(* CoDeSys 2.3.9.42 project: GLX_VCU_v3.3.0.pro *)
(* Author: JvL *)
(* Libraries: ifm_RAWCan\ifm_RAWCan_NT_V020004.lib 7.6.24 16:48:07, ifm_CR0403\ifm_CR0403_V030400.lib 31.5.24 17:04:27, ifm_CANopen\ifm_NetVarLib_NT_V020004.lib 7.6.24 16:46:42, standard.lib 4.10.05 11:14:46, SysLibCallback.lib 7.6.24 16:43:25, 3S_CANOPENNETVAR.LIB 7.6.24 16:46:41, Iecsfc.lib 13.4.06 15:51:28, Util.lib 7.6.24 16:43:26, ifm_CANopen\3S_CANopenManager.lib 7.6.24 16:46:41, ifm_CANopen\3S_CanDrv.lib 7.6.24 16:46:41 *)

(* PLC configuration (modules and I/O channels)
Configuration [LocalConfiguration] node 0, in %IB0 out %QB0 {IFM_PARAM_WORD_TIME = 0}
AT %IB0 [ChInputBool] Input 00 Bit
AT %IB1 [ChInputBool] Input 01 Bit
AT %IB2 [ChInputBool] Input 02 Bit
AT %IB3 [ChInputBool] Input 03 Bit
IGNITION_KEY AT %IB4 [ChInputBool] Input 04 Bit
CHARGER_INPUT AT %IB5 [ChInputBool] Input 05 Bit
BATTERY1_IGNITION AT %IB6 [ChInputBool] Input 06 Bit
BATTERY2_IGNITION AT %IB7 [ChInputBool] Input 07 Bit
ARM_SWITCH AT %IB8 [ChInputBool] Input 08 Bit
KILL_SWITCH AT %IB9 [ChInputBool] Input 09 Bit
HYDRAULIC_SWITCH AT %IB10 [ChInputBool] Input 10 Bit
EM_SWITCH AT %IB11 [ChInputBool] Input 11 Bit
ARM_LED AT %QB0 [ChOutputBool] Output 00 Bit
PRECHARGE_RELAY AT %QB1 [ChOutputBool] Output 01 Bit
AT %QB2 [ChOutputBool] Output 02 Bit
BRAKE_LIGHT AT %QB3 [ChOutputBool] Output 03 Bit
EM_BRAKE AT %QB4 [ChOutputBool] Output 04 Bit
MCU_IGNITION AT %QB5 [ChOutputBool] Output 05 Bit
BATTERY1_RELAY AT %QB6 [ChOutputBool] Output 06 Bit
BATTERY2_RELAY AT %QB7 [ChOutputBool] Output 07 Bit
HORN AT %QB8 [ChOutputBool] Output 08 Bit
BUZZER AT %QB9 [ChOutputBool] Output 09 Bit
CONTACTOR AT %QB10 [ChOutputBool] Output 10 Bit
CHARGING_LED AT %QB11 [ChOutputBool] Output 11 Bit
System Inputs [LocalSystemInputs] node 2, in %IB12 out %QB12
  SUPPLY_VOLTAGE_VBBS AT %IW6 [ChInputWord] Supply voltage VBBS
  SUPPLY_VOLTAGE_VU AT %IW7 [ChInputWord] Supply voltage VU
  SUPPLY_VOLTAGE_VBB1 AT %IW8 [ChInputWord] Supply voltage VBB1
  SUPPLY_VOLTAGE_VBB2 AT %IW9 [ChInputWord] Supply voltage VBB2
  TEMPERATURE AT %IW10 [ChInputInt] Temperature
J1939 Interface [CAN_J1939] node 1, in %IB37 out %QB12
Interface CAN 2 [CAN_BUS] node 1, in %IB37 out %QB12 {STACK_DWORD_S = 0}
  J1939 Interface [CAN_J1939] node 1, in %IB37 out %QB12
*)

(* Global variable list: CanOpen implicit Variables *)
VAR_GLOBAL CONSTANT
	MAX_CTRLINDEX : INT := 0;
END_VAR

(* Global variable list: Global_Variables *)
VAR_GLOBAL
(*BATTERY*)
	BATTERY1_SOC: BYTE;
	BATTERY1_SOH: BYTE;
	BATTERY1_CHARGING: BOOL;
	BATTERY1_POWER: INT;
	BATTERY1_NTC1: BYTE;
	BATTERY1_NTC2: BYTE;
	BATTERY1_CAN_ERROR: BOOL;
	BATTERY1_CAPACITY: INT;
	BATTERY1_TOTAL_CAPACITY: INT;
	BATTERY1_CURRENT: INT;
	BATTERY1_FULLCHARGE_MIN: REAL;

	BATTERY2_SOC: BYTE;
	BATTERY2_SOH: BYTE;
	BATTERY2_CHARGING: BOOL;
	BATTERY2_POWER: INT;
	BATTERY2_NTC1: BYTE;
	BATTERY2_NTC2: BYTE;
	BATTERY2_CAN_ERROR: BOOL;
	BATTERY2_CAPACITY: INT;
	BATTERY2_TOTAL_CAPACITY: INT;
	BATTERY2_CURRENT: INT;
	BATTERY2_FULLCHARGE_MIN: REAL;

(*MCU <> MOTOR*)
	MOTOR_TARGET_RPM: ARRAY [1..6] OF INT;
	MOTOR_IGNITION: ARRAY [1..6] OF BOOL;

	MOTOR_RPM: ARRAY [1..6] OF INT;
	MOTOR_POWER: ARRAY [1..6] OF INT;
	MOTOR_PHASE_CURRENT: ARRAY [1..6] OF WORD;
	MOTOR_TEMPERATURE:ARRAY [1..6] OF BYTE;
	MCU_TEMPERATURE:ARRAY [1..6] OF BYTE;
	MCU_CAN_ERROR: ARRAY [1..6] OF BOOL;

	MOTOR1_FAULT_ARRAY: ARRAY [1..4] OF BYTE;
	MOTOR2_FAULT_ARRAY: ARRAY [1..4] OF BYTE;
	MOTOR6_FAULT_ARRAY: ARRAY [1..4] OF BYTE;
       MOTOR_OBD_ARRAY: ARRAY [1..6] OF WORD;

(*JOYSTICK*)
	LOG_JX: BYTE;
	LOG_JY: BYTE;
	JOY_ERROR: BOOL;
(*IMU*)
	X_ANGLE_BYTE:BYTE;
	Y_ANGLE_BYTE:BYTE;
	NEG_Y: BOOL;
	NEG_X: BOOL;
	Y_MAX_PEAK: BYTE;
	X_MAX_PEAK: BYTE;
	Y_MIN_PEAK: BYTE;
	X_MIN_PEAK: BYTE;
	IMU_CAN_ERROR:BOOL;
	IMU_ALERT: BOOL;
(*DISPLAY TELEMATICS*)
	HIGH_SPEED: BOOL;
	POWER_MODE: BOOL;
	HILL_HOLD: BOOL;
	DISABLE_MCU_CAN: BOOL;
	TRIP_RESET: BOOL;
      	BATTERY_CHARGING:BOOL;
(*MISC*)
	REVERSE: BOOL;
	MCU_BRAKE: BOOL;
(*HYDRAULICS*)
	HYDRAULIC_IGNITION: BOOL;
(*CALCULATIONS*)
	AVG_RPM: INT;
	RANGE_IN_KM: BYTE;
	SPEED: BYTE;

	RUNTIME: DWORD;
	HYDL_UP_TIME:DWORD;
	VEHICLE_UP_TIME: DWORD;
	VEHICLE_UP_TIME_LT: DWORD;

	ODO_KM: WORD;
	ODO_METER: DWORD;

	TRIP_METER: DWORD;
	TRIP_KM: WORD;

	DUMMY: BOOL;
END_VAR
VAR_GLOBAL RETAIN
	Y_MAX_RETAIN: BYTE;
	X_MAX_RETAIN: BYTE;
	Y_MIN_RETAIN: BYTE;
	X_MIN_RETAIN: BYTE;
END_VAR

(* Global variable list: Networkmanagement implicit Variables CAN *)
VAR_GLOBAL CONSTANT
	USE_NWVARS_CAN : BOOL := FALSE;
	MAX_NetVarItems_CAN	: INT := 0;
	MAX_NetVarPDO_Rx_CAN	: INT := 0;
	MAX_NetVarPDO_Tx_CAN	: INT := 0;
	MAX_NetVarOD_CAN		: INT := 0;
END_VAR
VAR_GLOBAL
	pNetVarItems_CAN		: ARRAY[0..MAX_NetVarItems_CAN] OF NetVarDataItem_CAN;
	pNetVarPDO_Rx_CAN		: ARRAY[0..MAX_NetVarPDO_Rx_CAN] OF NetVarPDO_Rx_CAN;
	pNetVarPDO_Tx_CAN		: ARRAY[0..MAX_NetVarPDO_Tx_CAN] OF NetVarPDO_Tx_CAN;
	pNetVarOD_CAN			: ARRAY[0..MAX_NetVarOD_CAN] OF NetVarOD_CAN;
END_VAR

(* POU PLC_PRG, FBD *)
PROGRAM PLC_PRG
VAR
	CONTACTOR_DELAY: TON;
END_VAR
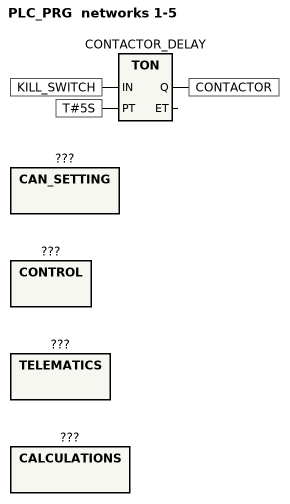
_FBD_ (* Function Block Diagram *)
NETWORK 1
	CONTACTOR_DELAY:TON(IN: KILL_SWITCH, PT: T#5S) => CONTACTOR
NETWORK 2
	???:CAN_SETTING()
NETWORK 3
	???:CONTROL()
NETWORK 4
	???:TELEMATICS()
NETWORK 5
	???:CALCULATIONS()
_END_FBD_
(* the same logic as Structured Text *)
(* Network 1 *)
CONTACTOR_DELAY(IN := KILL_SWITCH, PT := T#5S);
CONTACTOR := CONTACTOR_DELAY.Q;
(* Network 2: see the listing above *)
(* Network 3: see the listing above *)
(* Network 4: see the listing above *)
(* Network 5: see the listing above *)
END_PROGRAM

(* POU CAN_SETTING/CAN_SETTING, FBD *)
PROGRAM CAN_SETTING
(*
Created By: BHAGYESH
Date: 20-01-2024
Version: 1
Description: This program enables the CAN channels and sets the basic CAN parameter for both channels.
This block also controls the IFM's Inbuilt LED.
*)
VAR
	CAN_EN_1: CAN_ENABLE;
	CAN_EN_2: CAN_ENABLE;
	CAN_SET_1: CAN_SETDOWNLOADID;
	CAN_SET_2: CAN_SETDOWNLOADID;
	LED_SET: SET_LED;
	CAN_STATUS_1: CAN_STATUS;
	CAN_STATUS_2: CAN_STATUS;
	RESET_1: BOOL;
	RESET_2: BOOL;
END_VAR
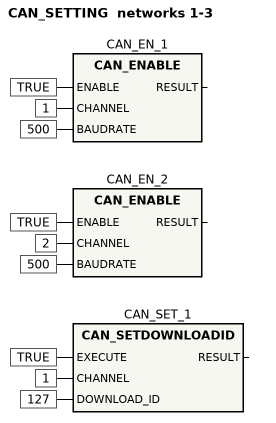
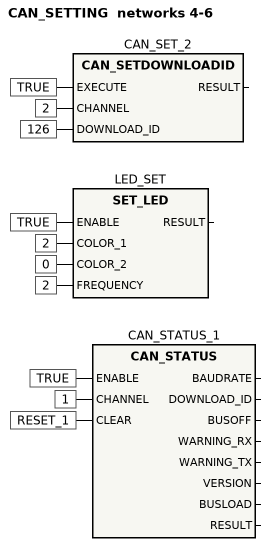
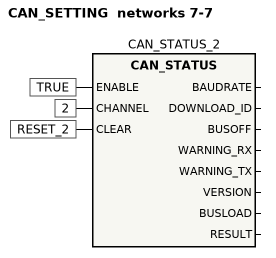
_FBD_ (* Function Block Diagram *)
NETWORK 1
	CAN_EN_1:CAN_ENABLE(ENABLE: TRUE, CHANNEL: 1, BAUDRATE: 500)
NETWORK 2
	CAN_EN_2:CAN_ENABLE(ENABLE: TRUE, CHANNEL: 2, BAUDRATE: 500)
NETWORK 3
	CAN_SET_1:CAN_SETDOWNLOADID(EXECUTE: TRUE, CHANNEL: 1, DOWNLOAD_ID: 127)
NETWORK 4
	CAN_SET_2:CAN_SETDOWNLOADID(EXECUTE: TRUE, CHANNEL: 2, DOWNLOAD_ID: 126)
NETWORK 5
	LED_SET:SET_LED(ENABLE: TRUE, COLOR_1: 2, COLOR_2: 0, FREQUENCY: 2)
NETWORK 6
	CAN_STATUS_1:CAN_STATUS(ENABLE: TRUE, CHANNEL: 1, CLEAR: RESET_1)
NETWORK 7
	CAN_STATUS_2:CAN_STATUS(ENABLE: TRUE, CHANNEL: 2, CLEAR: RESET_2)
_END_FBD_
(* the same logic as Structured Text *)
(* Network 1 *)
CAN_EN_1(ENABLE := TRUE, CHANNEL := 1, BAUDRATE := 500);
(* Network 2 *)
CAN_EN_2(ENABLE := TRUE, CHANNEL := 2, BAUDRATE := 500);
(* Network 3 *)
CAN_SET_1(EXECUTE := TRUE, CHANNEL := 1, DOWNLOAD_ID := 127);
(* Network 4 *)
CAN_SET_2(EXECUTE := TRUE, CHANNEL := 2, DOWNLOAD_ID := 126);
(* Network 5 *)
LED_SET(ENABLE := TRUE, COLOR_1 := 2, COLOR_2 := 0, FREQUENCY := 2);
(* Network 6 *)
CAN_STATUS_1(ENABLE := TRUE, CHANNEL := 1, CLEAR := RESET_1);
(* Network 7 *)
CAN_STATUS_2(ENABLE := TRUE, CHANNEL := 2, CLEAR := RESET_2);
END_PROGRAM

(* POU CONTROL, LD *)
PROGRAM CONTROL
(*
CH1 (500KBPS) :  MAKERSAN JOYSTICK								CH2 (500KBPS):	CLN BATTERY1
					DWIN DISPLAY															CLN BATTERY2
					BYTEBEAM  &  TOR														CHARA MCU 1
					MAKESAN IMU															CHARA MCU 2	
																								CHARA MCU 3
																								SOLTERRA CHARGER
			***UPDATES***
> Visualization update
> Chara can tx block updated
> Actual rpm of tx block changed to reference rpm
>Updated AVG_RPM in tx block input.
> MAKERSAN Joystick added
>RPM FACTOR IS 40 for 4000 RPM
> Battery channel changed and ramp decreased
>BATTERY CHARGING 
>MCU HIGH TEMP CUTOFF
>SALERI PUMP 
>HIGH SPEED AND HORN BUTTON INVRTED

>The MCU has min ramp time of 100ms.
*)
VAR
	BATTERY: CLN_BATTERY;
	BATTERY_SELECTION: CLN_BATTERY_SELECTION;
	AUTO_CHARGING: CLN_CHARGING;

	JOYSTICK: MAKERSAN_JOYSTICK;
	ALT_SPEED: ALTERNATE;
	IMU: IMU_SENSOR;
	HYDRAULICS: HYDRAULIC_CONTROL;
	ARM: ARM_LOGIC;

	DRIVE: DRIVE_LOGIC;
	THROTTLE: THROTTLE_LOGIC;
	THROTTLE_RIGHT: INT;
	THROTTLE_LEFT: INT;

	MCU_TX_RIGHT: CHARA_MCU_TX;
	MCU_TX_LEFT: CHARA_MCU_TX;
	MCU_RX_RIGHT: CHARA_MCU_RX;
	MCU_RX_LEFT: CHARA_MCU_RX;

	SALERI_PUMP: PWM1000;
	COOLANT_PUMP_ON: BOOL;
      VAL:WORD;

	RIGHT_ZERO: BOOL;
	LEFT_ZERO: BOOL;
	POWER_ZERO: BOOL;

	TEMP_CUTOFF: BOOL;
	MCU_HIGH_TEMP: BOOL;
	MCU_LOW_TEMP: BOOL;

	LOW5_SOC: BOOL;
	LOW20_SOC: BOOL;
	LOW_SOC: F_TRIG;
	LOW_SOC_TIMER: TP;
	LOWSOC_BLINK: BLINK;

	IMU_BLINK: BLINK;
	REVERSE_BLINK: BLINK;
	CHARGE_ERROR_BLINK: BLINK;
       LOW_SOC_BUZZER: BOOL;

	RX_227: RX_CAN;
	TOF_227: TOF;
	CHARGER_5kW_INPUT: BOOL;
	CHARGING_5KW: CAN_TX;

	CHARGE_ERROR_LIGHT: BLINK;
	DDD: BOOL;
	STARTING_BLINK: BLINK;
	OVER_TEMP_BLINK: BLINK;
END_VAR
VAR CONSTANT
	RPM_FACTOR: INT := 45;
	RAMP: INT:= 1000;
	MCU_RAMP: BYTE := 8;
	PHASE_LIMIT: BYTE := 60;
	CHARGING_FRAME: ARRAY [0..7] OF BYTE := 16#03, 16#25, 16#01, 16#90, 0, 0, 0, 0;
END_VAR
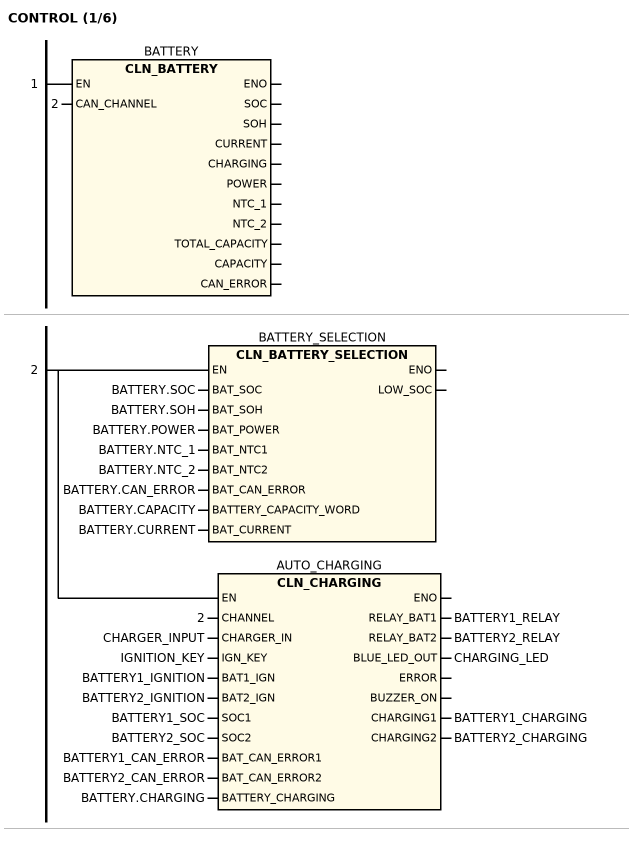
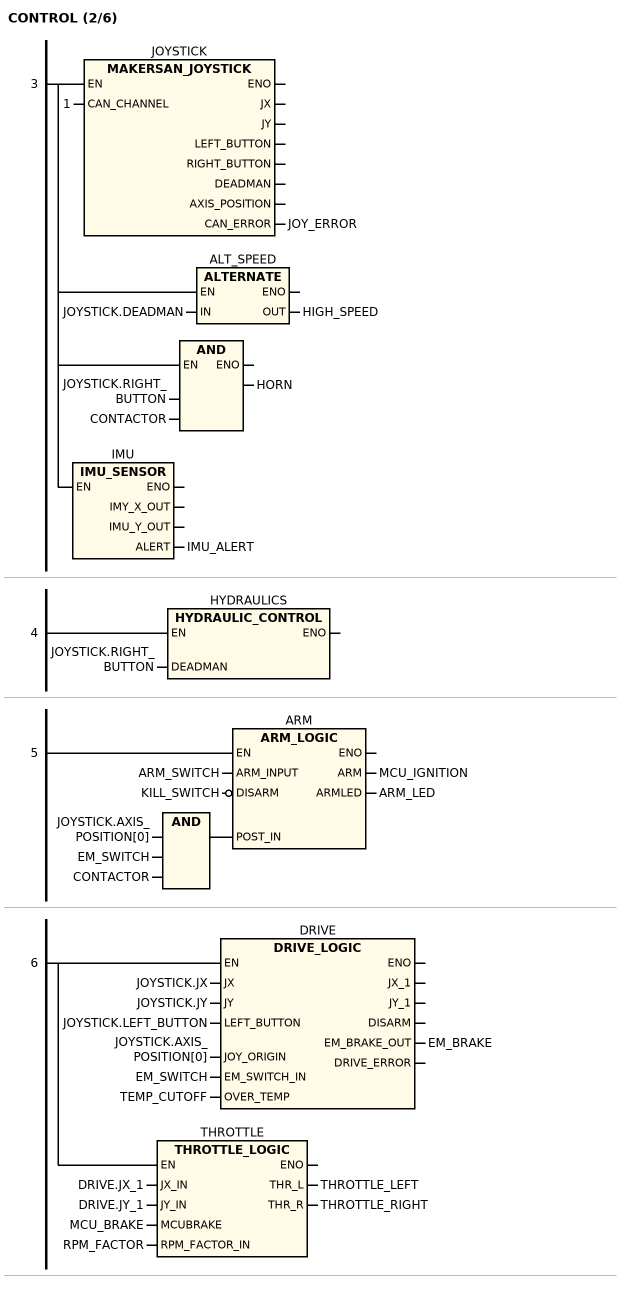
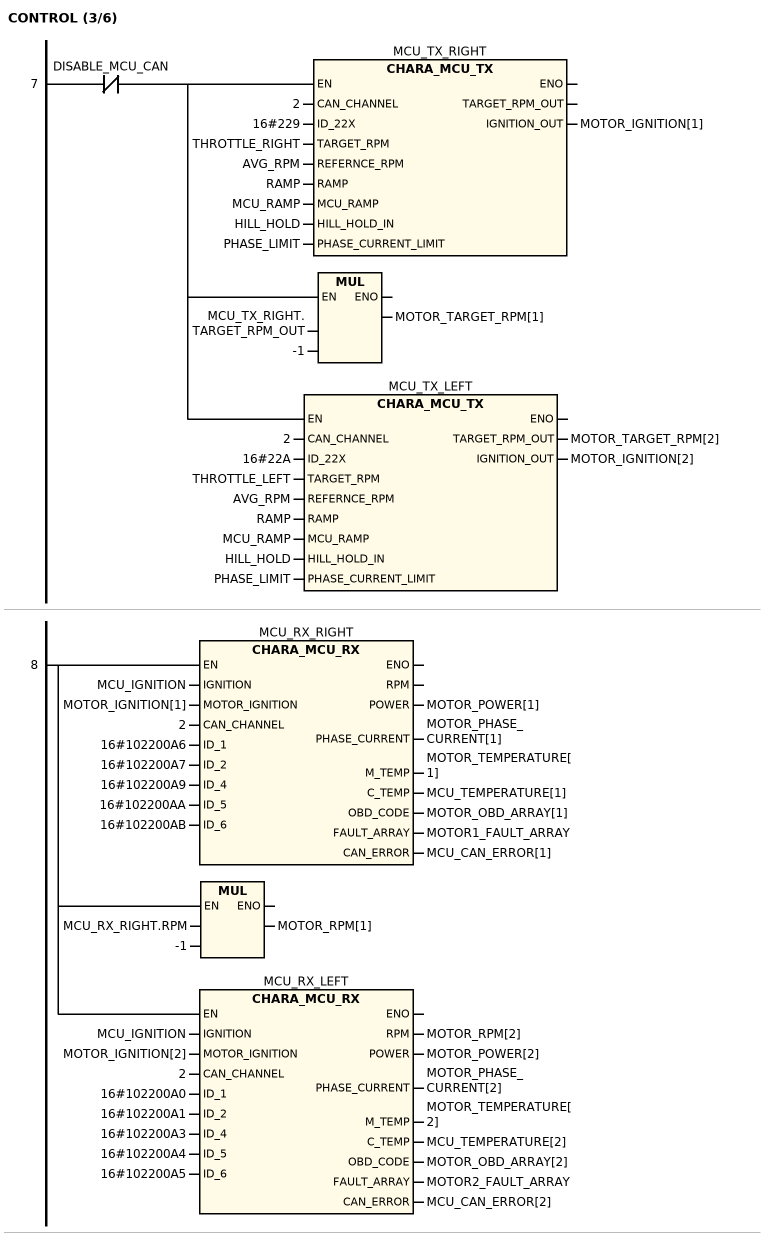
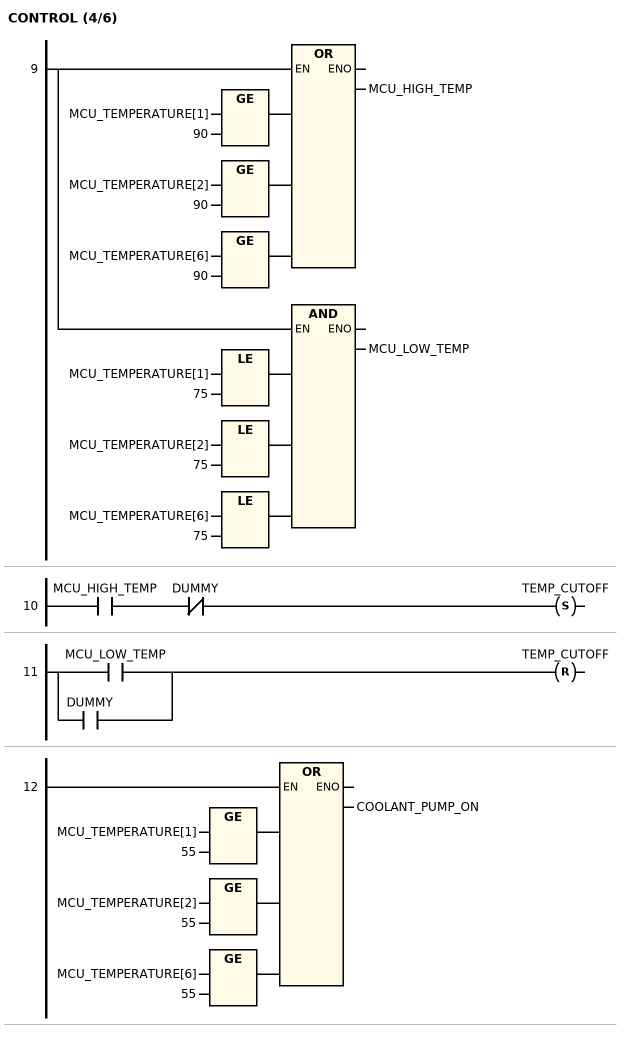
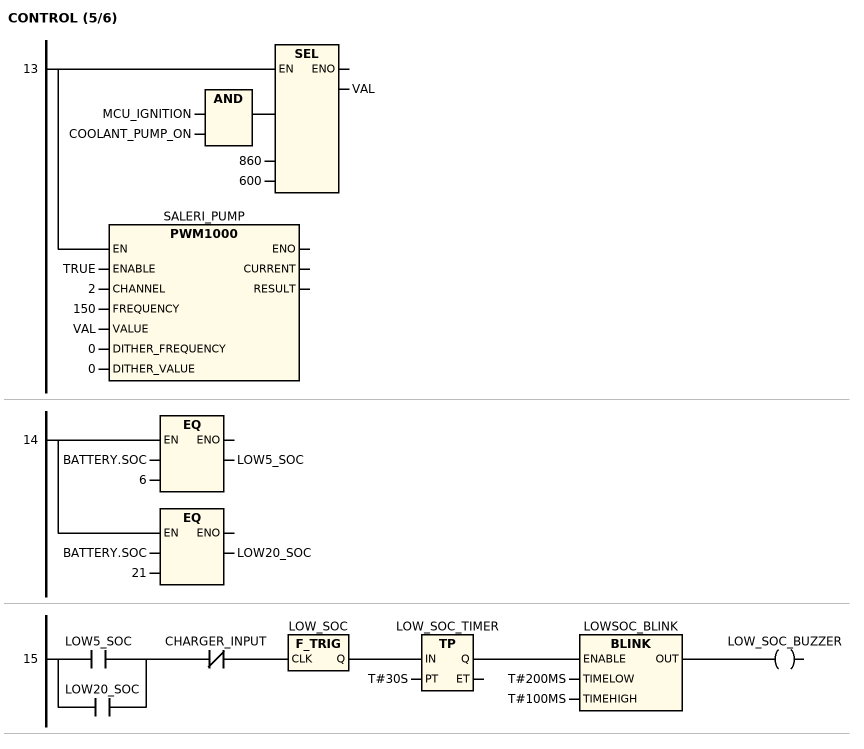
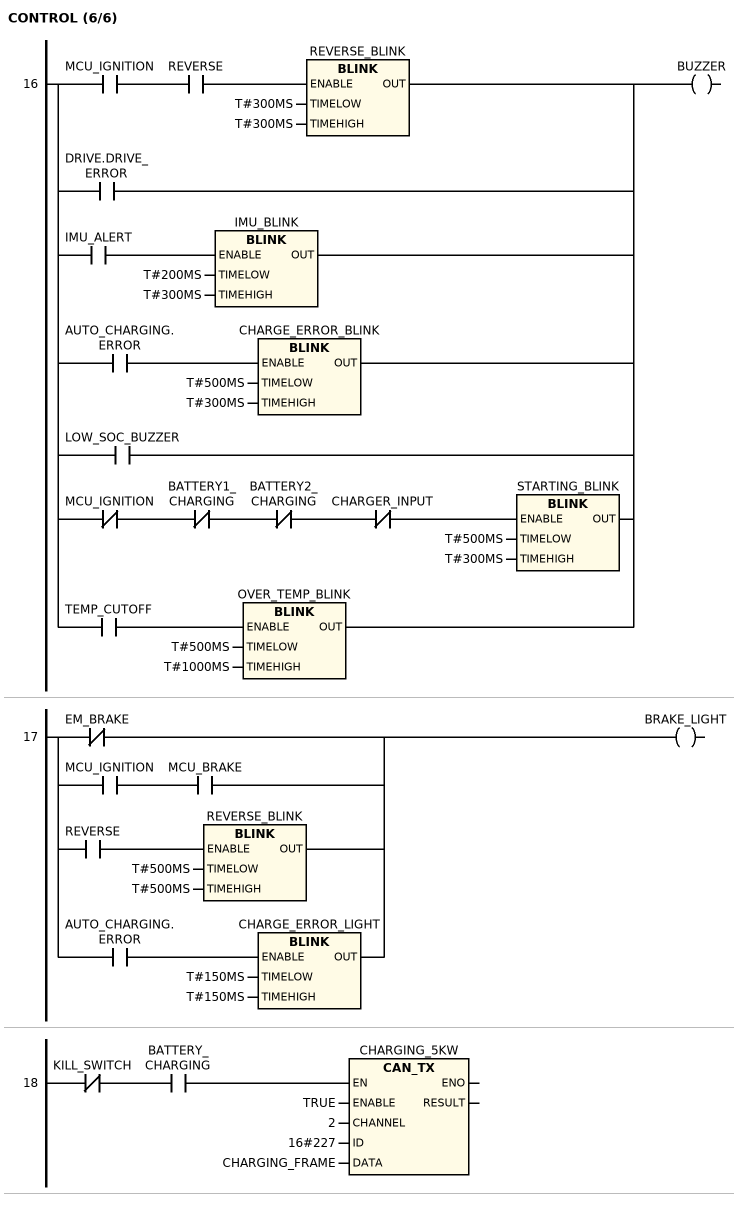
_LD_ (* Ladder Diagram *)
NETWORK 1
	*
		EN --- BATTERY:CLN_BATTERY(CAN_CHANNEL: 2)
NETWORK 2
	*
		EN --- BATTERY_SELECTION:CLN_BATTERY_SELECTION(BAT_SOC: BATTERY.SOC, BAT_SOH: BATTERY.SOH, BAT_POWER: BATTERY.POWER, BAT_NTC1: BATTERY.NTC_1, BAT_NTC2: BATTERY.NTC_2, BAT_CAN_ERROR: BATTERY.CAN_ERROR, BATTERY_CAPACITY_WORD: BATTERY.CAPACITY, BAT_CURRENT: BATTERY.CURRENT)
		EN --- AUTO_CHARGING:CLN_CHARGING(CHANNEL: 2, CHARGER_IN: CHARGER_INPUT, IGN_KEY: IGNITION_KEY, BAT1_IGN: BATTERY1_IGNITION, BAT2_IGN: BATTERY2_IGNITION, SOC1: BATTERY1_SOC, SOC2: BATTERY2_SOC, BAT_CAN_ERROR1: BATTERY1_CAN_ERROR, BAT_CAN_ERROR2: BATTERY2_CAN_ERROR, BATTERY_CHARGING: BATTERY.CHARGING, RELAY_BAT2 => BATTERY2_RELAY, BLUE_LED_OUT => CHARGING_LED, CHARGING1 => BATTERY1_CHARGING, CHARGING2 => BATTERY2_CHARGING) => BATTERY1_RELAY
NETWORK 3
	*
		EN --- JOYSTICK:MAKERSAN_JOYSTICK(CAN_CHANNEL: 1, CAN_ERROR => JOY_ERROR)
		EN --- ALT_SPEED:ALTERNATE(IN: JOYSTICK.DEADMAN) => HIGH_SPEED
		EN --- AND(JOYSTICK.RIGHT_BUTTON, CONTACTOR) => HORN
		EN --- IMU:IMU_SENSOR(ALERT => IMU_ALERT)
NETWORK 4
	*
		EN --- HYDRAULICS:HYDRAULIC_CONTROL(DEADMAN: JOYSTICK.RIGHT_BUTTON)
NETWORK 5
	*
		EN --- ARM:ARM_LOGIC(ARM_INPUT: ARM_SWITCH, DISARM: NOT KILL_SWITCH, POST_IN: AND(JOYSTICK.AXIS_POSITION[0], EM_SWITCH, CONTACTOR), ARMLED => ARM_LED) => MCU_IGNITION
NETWORK 6
	*
		EN --- DRIVE:DRIVE_LOGIC(JX: JOYSTICK.JX, JY: JOYSTICK.JY, LEFT_BUTTON: JOYSTICK.LEFT_BUTTON, JOY_ORIGIN: JOYSTICK.AXIS_POSITION[0], EM_SWITCH_IN: EM_SWITCH, OVER_TEMP: TEMP_CUTOFF, EM_BRAKE_OUT => EM_BRAKE)
		EN --- THROTTLE:THROTTLE_LOGIC(JX_IN: DRIVE.JX_1, JY_IN: DRIVE.JY_1, MCUBRAKE: MCU_BRAKE, RPM_FACTOR_IN: RPM_FACTOR, THR_R => THROTTLE_RIGHT) => THROTTLE_LEFT
NETWORK 7
	[/DISABLE_MCU_CAN]
		EN --- MCU_TX_RIGHT:CHARA_MCU_TX(CAN_CHANNEL: 2, ID_22X: 16#229, TARGET_RPM: THROTTLE_RIGHT, REFERNCE_RPM: AVG_RPM, RAMP: RAMP, MCU_RAMP: MCU_RAMP, HILL_HOLD_IN: HILL_HOLD, PHASE_CURRENT_LIMIT: PHASE_LIMIT, IGNITION_OUT => MOTOR_IGNITION[1])
		EN --- MUL(MCU_TX_RIGHT.TARGET_RPM_OUT, -1) => MOTOR_TARGET_RPM[1]
		EN --- MCU_TX_LEFT:CHARA_MCU_TX(CAN_CHANNEL: 2, ID_22X: 16#22A, TARGET_RPM: THROTTLE_LEFT, REFERNCE_RPM: AVG_RPM, RAMP: RAMP, MCU_RAMP: MCU_RAMP, HILL_HOLD_IN: HILL_HOLD, PHASE_CURRENT_LIMIT: PHASE_LIMIT, IGNITION_OUT => MOTOR_IGNITION[2]) => MOTOR_TARGET_RPM[2]
NETWORK 8
	*
		EN --- MCU_RX_RIGHT:CHARA_MCU_RX(IGNITION: MCU_IGNITION, MOTOR_IGNITION: MOTOR_IGNITION[1], CAN_CHANNEL: 2, ID_1: 16#102200A6, ID_2: 16#102200A7, ID_4: 16#102200A9, ID_5: 16#102200AA, ID_6: 16#102200AB, POWER => MOTOR_POWER[1], PHASE_CURRENT => MOTOR_PHASE_CURRENT[1], M_TEMP => MOTOR_TEMPERATURE[1], C_TEMP => MCU_TEMPERATURE[1], OBD_CODE => MOTOR_OBD_ARRAY[1], FAULT_ARRAY => MOTOR1_FAULT_ARRAY, CAN_ERROR => MCU_CAN_ERROR[1])
		EN --- MUL(MCU_RX_RIGHT.RPM, -1) => MOTOR_RPM[1]
		EN --- MCU_RX_LEFT:CHARA_MCU_RX(IGNITION: MCU_IGNITION, MOTOR_IGNITION: MOTOR_IGNITION[2], CAN_CHANNEL: 2, ID_1: 16#102200A0, ID_2: 16#102200A1, ID_4: 16#102200A3, ID_5: 16#102200A4, ID_6: 16#102200A5, POWER => MOTOR_POWER[2], PHASE_CURRENT => MOTOR_PHASE_CURRENT[2], M_TEMP => MOTOR_TEMPERATURE[2], C_TEMP => MCU_TEMPERATURE[2], OBD_CODE => MOTOR_OBD_ARRAY[2], FAULT_ARRAY => MOTOR2_FAULT_ARRAY, CAN_ERROR => MCU_CAN_ERROR[2]) => MOTOR_RPM[2]
NETWORK 9
	*
		EN --- OR(GE(MCU_TEMPERATURE[1], 90), GE(MCU_TEMPERATURE[2], 90), GE(MCU_TEMPERATURE[6], 90)) => MCU_HIGH_TEMP
		EN --- AND(LE(MCU_TEMPERATURE[1], 75), LE(MCU_TEMPERATURE[2], 75), LE(MCU_TEMPERATURE[6], 75)) => MCU_LOW_TEMP
NETWORK 10
	[MCU_HIGH_TEMP] - [/DUMMY] --- (S TEMP_CUTOFF)
NETWORK 11
	{ [MCU_LOW_TEMP] | [DUMMY] } --- (R TEMP_CUTOFF)
NETWORK 12
	*
		EN --- OR(GE(MCU_TEMPERATURE[1], 55), GE(MCU_TEMPERATURE[2], 55), GE(MCU_TEMPERATURE[6], 55)) => COOLANT_PUMP_ON
NETWORK 13
	*
		EN --- SEL(AND(MCU_IGNITION, COOLANT_PUMP_ON), 860, 600) => VAL
		EN --- SALERI_PUMP:PWM1000(ENABLE: TRUE, CHANNEL: 2, FREQUENCY: 150, VALUE: VAL, DITHER_FREQUENCY: 0, DITHER_VALUE: 0)
NETWORK 14
	*
		EN --- EQ(BATTERY.SOC, 6) => LOW5_SOC
		EN --- EQ(BATTERY.SOC, 21) => LOW20_SOC
NETWORK 15
	{ [LOW5_SOC] | [LOW20_SOC] } - [/CHARGER_INPUT] - LOW_SOC:F_TRIG(CLK: *) - LOW_SOC_TIMER:TP(IN: *, PT: T#30S) - LOWSOC_BLINK:BLINK(ENABLE: *, TIMELOW: T#200MS, TIMEHIGH: T#100MS) --- (LOW_SOC_BUZZER)
NETWORK 16
	{ [MCU_IGNITION] - [REVERSE] - REVERSE_BLINK:BLINK(ENABLE: *, TIMELOW: T#300MS, TIMEHIGH: T#300MS) | [DRIVE.DRIVE_ERROR] | [IMU_ALERT] - IMU_BLINK:BLINK(ENABLE: *, TIMELOW: T#200MS, TIMEHIGH: T#300MS) | [AUTO_CHARGING.ERROR] - CHARGE_ERROR_BLINK:BLINK(ENABLE: *, TIMELOW: T#500MS, TIMEHIGH: T#300MS) | [LOW_SOC_BUZZER] | [/MCU_IGNITION] - [/BATTERY1_CHARGING] - [/BATTERY2_CHARGING] - [/CHARGER_INPUT] - STARTING_BLINK:BLINK(ENABLE: *, TIMELOW: T#500MS, TIMEHIGH: T#300MS) | [TEMP_CUTOFF] - OVER_TEMP_BLINK:BLINK(ENABLE: *, TIMELOW: T#500MS, TIMEHIGH: T#1000MS) } --- (BUZZER)
NETWORK 17
	{ [/EM_BRAKE] | [MCU_IGNITION] - [MCU_BRAKE] | [REVERSE] - REVERSE_BLINK:BLINK(ENABLE: *, TIMELOW: T#500MS, TIMEHIGH: T#500MS) | [AUTO_CHARGING.ERROR] - CHARGE_ERROR_LIGHT:BLINK(ENABLE: *, TIMELOW: T#150MS, TIMEHIGH: T#150MS) } --- (BRAKE_LIGHT)
NETWORK 18
	[/KILL_SWITCH] - [BATTERY_CHARGING]
		EN --- CHARGING_5KW:CAN_TX(ENABLE: TRUE, CHANNEL: 2, ID: 16#227, DATA: CHARGING_FRAME)
_END_LD_
(* the same logic as Structured Text *)
(* Network 1 *)
BATTERY(CAN_CHANNEL := 2);
(* Network 2 *)
BATTERY_SELECTION(BAT_SOC := BATTERY.SOC, BAT_SOH := BATTERY.SOH, BAT_POWER := BATTERY.POWER, BAT_NTC1 := BATTERY.NTC_1, BAT_NTC2 := BATTERY.NTC_2, BAT_CAN_ERROR := BATTERY.CAN_ERROR, BATTERY_CAPACITY_WORD := BATTERY.CAPACITY, BAT_CURRENT := BATTERY.CURRENT);
AUTO_CHARGING(CHANNEL := 2, CHARGER_IN := CHARGER_INPUT, IGN_KEY := IGNITION_KEY, BAT1_IGN := BATTERY1_IGNITION, BAT2_IGN := BATTERY2_IGNITION, SOC1 := BATTERY1_SOC, SOC2 := BATTERY2_SOC, BAT_CAN_ERROR1 := BATTERY1_CAN_ERROR, BAT_CAN_ERROR2 := BATTERY2_CAN_ERROR, BATTERY_CHARGING := BATTERY.CHARGING);
BATTERY2_RELAY := AUTO_CHARGING.RELAY_BAT2;
CHARGING_LED := AUTO_CHARGING.BLUE_LED_OUT;
BATTERY1_CHARGING := AUTO_CHARGING.CHARGING1;
BATTERY2_CHARGING := AUTO_CHARGING.CHARGING2;
BATTERY1_RELAY := AUTO_CHARGING.RELAY_BAT1;
(* Network 3 *)
JOYSTICK(CAN_CHANNEL := 1);
JOY_ERROR := JOYSTICK.CAN_ERROR;
ALT_SPEED(IN := JOYSTICK.DEADMAN);
HIGH_SPEED := ALT_SPEED.OUT;
HORN := JOYSTICK.RIGHT_BUTTON AND CONTACTOR;
IMU();
IMU_ALERT := IMU.ALERT;
(* Network 4 *)
HYDRAULICS(DEADMAN := JOYSTICK.RIGHT_BUTTON);
(* Network 5 *)
ARM(ARM_INPUT := ARM_SWITCH, DISARM := NOT KILL_SWITCH, POST_IN := JOYSTICK.AXIS_POSITION[0] AND EM_SWITCH AND CONTACTOR);
ARM_LED := ARM.ARMLED;
MCU_IGNITION := ARM.ARM;
(* Network 6 *)
DRIVE(JX := JOYSTICK.JX, JY := JOYSTICK.JY, LEFT_BUTTON := JOYSTICK.LEFT_BUTTON, JOY_ORIGIN := JOYSTICK.AXIS_POSITION[0], EM_SWITCH_IN := EM_SWITCH, OVER_TEMP := TEMP_CUTOFF);
EM_BRAKE := DRIVE.EM_BRAKE_OUT;
THROTTLE(JX_IN := DRIVE.JX_1, JY_IN := DRIVE.JY_1, MCUBRAKE := MCU_BRAKE, RPM_FACTOR_IN := RPM_FACTOR);
THROTTLE_RIGHT := THROTTLE.THR_R;
THROTTLE_LEFT := THROTTLE.THR_L;
(* Network 7 *)
IF NOT DISABLE_MCU_CAN THEN
	MCU_TX_RIGHT(CAN_CHANNEL := 2, ID_22X := 16#229, TARGET_RPM := THROTTLE_RIGHT, REFERNCE_RPM := AVG_RPM, RAMP := RAMP, MCU_RAMP := MCU_RAMP, HILL_HOLD_IN := HILL_HOLD, PHASE_CURRENT_LIMIT := PHASE_LIMIT);
	MOTOR_IGNITION[1] := MCU_TX_RIGHT.IGNITION_OUT;
	MOTOR_TARGET_RPM[1] := MCU_TX_RIGHT.TARGET_RPM_OUT * (-1);
	MCU_TX_LEFT(CAN_CHANNEL := 2, ID_22X := 16#22A, TARGET_RPM := THROTTLE_LEFT, REFERNCE_RPM := AVG_RPM, RAMP := RAMP, MCU_RAMP := MCU_RAMP, HILL_HOLD_IN := HILL_HOLD, PHASE_CURRENT_LIMIT := PHASE_LIMIT);
	MOTOR_IGNITION[2] := MCU_TX_LEFT.IGNITION_OUT;
	MOTOR_TARGET_RPM[2] := MCU_TX_LEFT.TARGET_RPM_OUT;
END_IF;
(* Network 8 *)
MCU_RX_RIGHT(IGNITION := MCU_IGNITION, MOTOR_IGNITION := MOTOR_IGNITION[1], CAN_CHANNEL := 2, ID_1 := 16#102200A6, ID_2 := 16#102200A7, ID_4 := 16#102200A9, ID_5 := 16#102200AA, ID_6 := 16#102200AB);
MOTOR_POWER[1] := MCU_RX_RIGHT.POWER;
MOTOR_PHASE_CURRENT[1] := MCU_RX_RIGHT.PHASE_CURRENT;
MOTOR_TEMPERATURE[1] := MCU_RX_RIGHT.M_TEMP;
MCU_TEMPERATURE[1] := MCU_RX_RIGHT.C_TEMP;
MOTOR_OBD_ARRAY[1] := MCU_RX_RIGHT.OBD_CODE;
MOTOR1_FAULT_ARRAY := MCU_RX_RIGHT.FAULT_ARRAY;
MCU_CAN_ERROR[1] := MCU_RX_RIGHT.CAN_ERROR;
MOTOR_RPM[1] := MCU_RX_RIGHT.RPM * (-1);
MCU_RX_LEFT(IGNITION := MCU_IGNITION, MOTOR_IGNITION := MOTOR_IGNITION[2], CAN_CHANNEL := 2, ID_1 := 16#102200A0, ID_2 := 16#102200A1, ID_4 := 16#102200A3, ID_5 := 16#102200A4, ID_6 := 16#102200A5);
MOTOR_POWER[2] := MCU_RX_LEFT.POWER;
MOTOR_PHASE_CURRENT[2] := MCU_RX_LEFT.PHASE_CURRENT;
MOTOR_TEMPERATURE[2] := MCU_RX_LEFT.M_TEMP;
MCU_TEMPERATURE[2] := MCU_RX_LEFT.C_TEMP;
MOTOR_OBD_ARRAY[2] := MCU_RX_LEFT.OBD_CODE;
MOTOR2_FAULT_ARRAY := MCU_RX_LEFT.FAULT_ARRAY;
MCU_CAN_ERROR[2] := MCU_RX_LEFT.CAN_ERROR;
MOTOR_RPM[2] := MCU_RX_LEFT.RPM;
(* Network 9 *)
MCU_HIGH_TEMP := (MCU_TEMPERATURE[1] >= 90) OR (MCU_TEMPERATURE[2] >= 90) OR (MCU_TEMPERATURE[6] >= 90);
MCU_LOW_TEMP := (MCU_TEMPERATURE[1] <= 75) AND (MCU_TEMPERATURE[2] <= 75) AND (MCU_TEMPERATURE[6] <= 75);
(* Network 10 *)
IF MCU_HIGH_TEMP AND NOT DUMMY THEN TEMP_CUTOFF := TRUE; END_IF;
(* Network 11 *)
IF MCU_LOW_TEMP OR DUMMY THEN TEMP_CUTOFF := FALSE; END_IF;
(* Network 12 *)
COOLANT_PUMP_ON := (MCU_TEMPERATURE[1] >= 55) OR (MCU_TEMPERATURE[2] >= 55) OR (MCU_TEMPERATURE[6] >= 55);
(* Network 13 *)
VAL := SEL(MCU_IGNITION AND COOLANT_PUMP_ON, 860, 600);
SALERI_PUMP(ENABLE := TRUE, CHANNEL := 2, FREQUENCY := 150, VALUE := VAL, DITHER_FREQUENCY := 0, DITHER_VALUE := 0);
(* Network 14 *)
LOW5_SOC := BATTERY.SOC = 6;
LOW20_SOC := BATTERY.SOC = 21;
(* Network 15 *)
LOW_SOC(CLK := (LOW5_SOC OR LOW20_SOC) AND NOT CHARGER_INPUT);
LOW_SOC_TIMER(IN := LOW_SOC.Q, PT := T#30S);
LOWSOC_BLINK(ENABLE := LOW_SOC_TIMER.Q, TIMELOW := T#200MS, TIMEHIGH := T#100MS);
LOW_SOC_BUZZER := LOWSOC_BLINK.OUT;
(* Network 16 *)
REVERSE_BLINK(ENABLE := MCU_IGNITION AND REVERSE, TIMELOW := T#300MS, TIMEHIGH := T#300MS);
IMU_BLINK(ENABLE := IMU_ALERT, TIMELOW := T#200MS, TIMEHIGH := T#300MS);
CHARGE_ERROR_BLINK(ENABLE := AUTO_CHARGING.ERROR, TIMELOW := T#500MS, TIMEHIGH := T#300MS);
STARTING_BLINK(ENABLE := NOT MCU_IGNITION AND NOT BATTERY1_CHARGING AND NOT BATTERY2_CHARGING AND NOT CHARGER_INPUT, TIMELOW := T#500MS, TIMEHIGH := T#300MS);
OVER_TEMP_BLINK(ENABLE := TEMP_CUTOFF, TIMELOW := T#500MS, TIMEHIGH := T#1000MS);
BUZZER := REVERSE_BLINK.OUT OR DRIVE.DRIVE_ERROR OR IMU_BLINK.OUT OR CHARGE_ERROR_BLINK.OUT OR LOW_SOC_BUZZER OR STARTING_BLINK.OUT OR OVER_TEMP_BLINK.OUT;
(* Network 17 *)
REVERSE_BLINK(ENABLE := REVERSE, TIMELOW := T#500MS, TIMEHIGH := T#500MS);
CHARGE_ERROR_LIGHT(ENABLE := AUTO_CHARGING.ERROR, TIMELOW := T#150MS, TIMEHIGH := T#150MS);
BRAKE_LIGHT := NOT EM_BRAKE OR MCU_IGNITION AND MCU_BRAKE OR REVERSE_BLINK.OUT OR CHARGE_ERROR_LIGHT.OUT;
(* Network 18 *)
IF NOT KILL_SWITCH AND BATTERY_CHARGING THEN
	CHARGING_5KW(ENABLE := TRUE, CHANNEL := 2, ID := 16#227, DATA := CHARGING_FRAME);
END_IF;
END_PROGRAM

(* POU PROGRAM_FBs/CLN_BATTERY, LD *)
FUNCTION_BLOCK CLN_BATTERY
(*
Created by: Anirudh Raghavan
Date: 10-01-24
Version: 4
Updated by: Bhagyesh
Update date: 15-09-2024
Description: This block reads the data of CLN Battery.
	
	*** UPDATES ***
V3: 
	Removed the SOC mapping function.
V4
	Variable modifiacations and faults removed
*)
VAR_INPUT
	CAN_CHANNEL: BYTE;
END_VAR
VAR_OUTPUT
	SOC: BYTE;
	SOH: BYTE;
       CURRENT: INT;
	CHARGING: BOOL;
	POWER: INT; (*Watt*)
	NTC_1: BYTE;
	NTC_2: BYTE;
	TOTAL_CAPACITY: INT; (*Ah*)
	CAPACITY: INT; (*Ah*)
	CAN_ERROR: BOOL;

END_VAR
VAR
	RX_205: RX_CAN;
	RX_1E1: RX_CAN;
	RX_1F5: RX_CAN;
	RX_357: RX_CAN;
	DELAY: TON;
	SOC_WORD: WORD;
	SOH_WORD: WORD;
	VOLTAGE_WORD: WORD;
	CURRENT_WORD: WORD;
	VOLTAGE: INT;
	CAPACITY_WORD: WORD;
	CAPACITY_AH: WORD;
	TOTAL_CAPACITY_WORD: WORD;
	TOTAL_CAPACITY_AH: WORD;

END_VAR
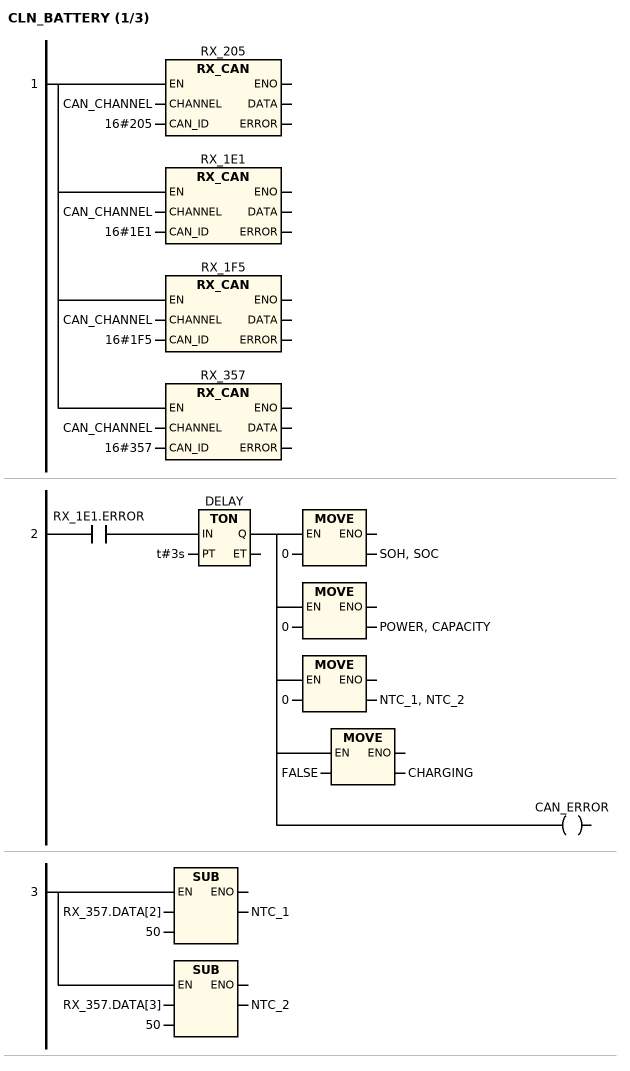
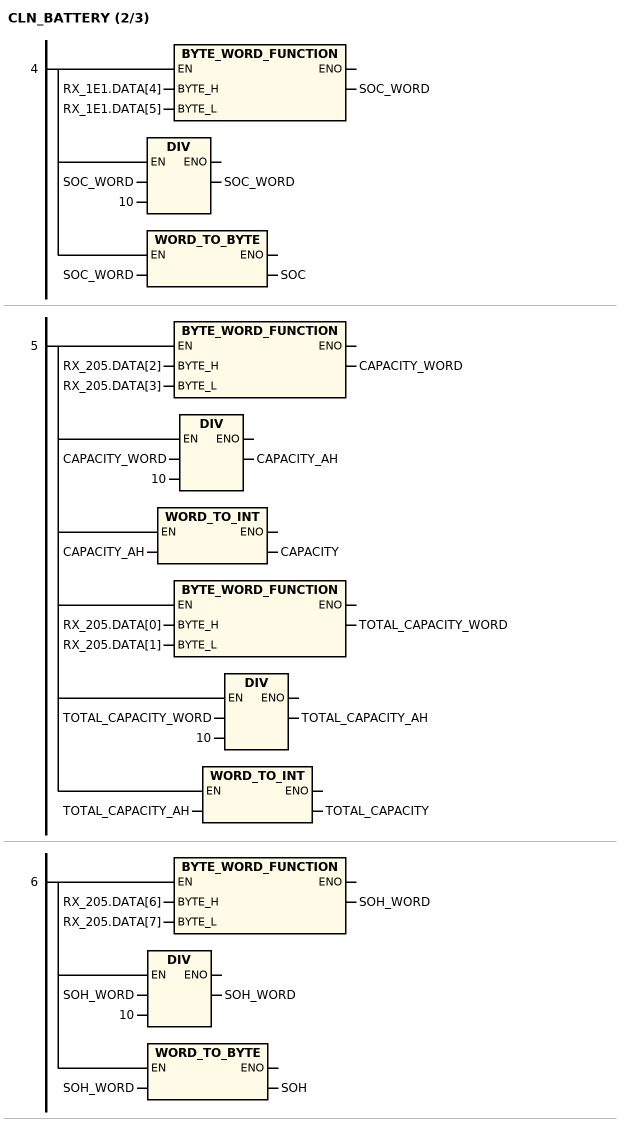
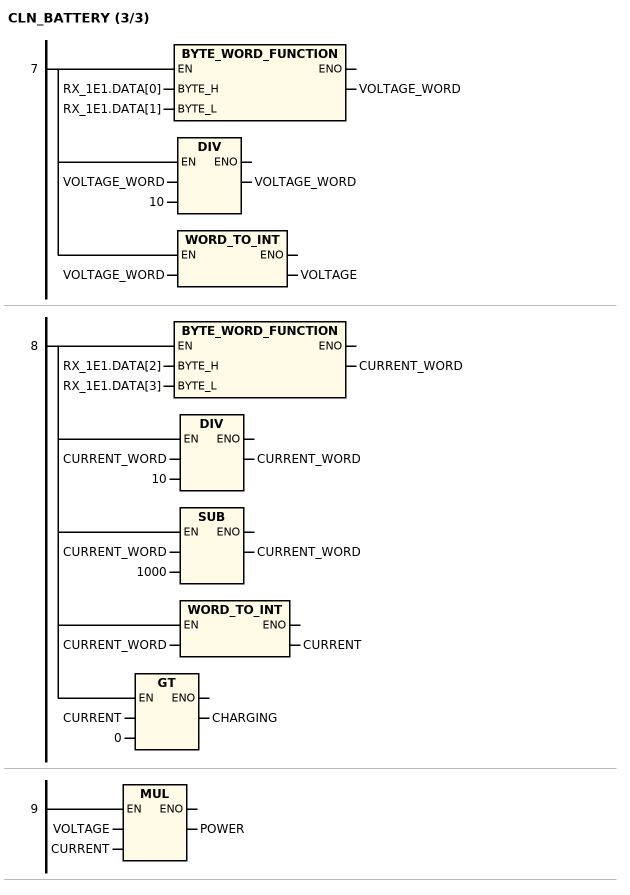
_LD_ (* Ladder Diagram *)
NETWORK 1
	*
		EN --- RX_205:RX_CAN(CHANNEL: CAN_CHANNEL, CAN_ID: 16#205)
		EN --- RX_1E1:RX_CAN(CHANNEL: CAN_CHANNEL, CAN_ID: 16#1E1)
		EN --- RX_1F5:RX_CAN(CHANNEL: CAN_CHANNEL, CAN_ID: 16#1F5)
		EN --- RX_357:RX_CAN(CHANNEL: CAN_CHANNEL, CAN_ID: 16#357)
NETWORK 2
	[RX_1E1.ERROR] - DELAY:TON(IN: *, PT: t#3s) --- (CAN_ERROR)
		EN --- MOVE(0) => SOH, SOC
		EN --- MOVE(0) => POWER, CAPACITY
		EN --- MOVE(0) => NTC_1, NTC_2
		EN --- MOVE(FALSE) => CHARGING
NETWORK 3
	*
		EN --- SUB(RX_357.DATA[2], 50) => NTC_1
		EN --- SUB(RX_357.DATA[3], 50) => NTC_2
NETWORK 4
	*
		EN --- BYTE_WORD_FUNCTION(BYTE_H: RX_1E1.DATA[4], BYTE_L: RX_1E1.DATA[5]) => SOC_WORD
		EN --- DIV(SOC_WORD, 10) => SOC_WORD
		EN --- WORD_TO_BYTE(SOC_WORD) => SOC
NETWORK 5
	*
		EN --- BYTE_WORD_FUNCTION(BYTE_H: RX_205.DATA[2], BYTE_L: RX_205.DATA[3]) => CAPACITY_WORD
		EN --- DIV(CAPACITY_WORD, 10) => CAPACITY_AH
		EN --- WORD_TO_INT(CAPACITY_AH) => CAPACITY
		EN --- BYTE_WORD_FUNCTION(BYTE_H: RX_205.DATA[0], BYTE_L: RX_205.DATA[1]) => TOTAL_CAPACITY_WORD
		EN --- DIV(TOTAL_CAPACITY_WORD, 10) => TOTAL_CAPACITY_AH
		EN --- WORD_TO_INT(TOTAL_CAPACITY_AH) => TOTAL_CAPACITY
NETWORK 6
	*
		EN --- BYTE_WORD_FUNCTION(BYTE_H: RX_205.DATA[6], BYTE_L: RX_205.DATA[7]) => SOH_WORD
		EN --- DIV(SOH_WORD, 10) => SOH_WORD
		EN --- WORD_TO_BYTE(SOH_WORD) => SOH
NETWORK 7
	*
		EN --- BYTE_WORD_FUNCTION(BYTE_H: RX_1E1.DATA[0], BYTE_L: RX_1E1.DATA[1]) => VOLTAGE_WORD
		EN --- DIV(VOLTAGE_WORD, 10) => VOLTAGE_WORD
		EN --- WORD_TO_INT(VOLTAGE_WORD) => VOLTAGE
NETWORK 8
	*
		EN --- BYTE_WORD_FUNCTION(BYTE_H: RX_1E1.DATA[2], BYTE_L: RX_1E1.DATA[3]) => CURRENT_WORD
		EN --- DIV(CURRENT_WORD, 10) => CURRENT_WORD
		EN --- SUB(CURRENT_WORD, 1000) => CURRENT_WORD
		EN --- WORD_TO_INT(CURRENT_WORD) => CURRENT
		EN --- GT(CURRENT, 0) => CHARGING
NETWORK 9
	*
		EN --- MUL(VOLTAGE, CURRENT) => POWER
_END_LD_
(* the same logic as Structured Text *)
(* Network 1 *)
RX_205(CHANNEL := CAN_CHANNEL, CAN_ID := 16#205);
RX_1E1(CHANNEL := CAN_CHANNEL, CAN_ID := 16#1E1);
RX_1F5(CHANNEL := CAN_CHANNEL, CAN_ID := 16#1F5);
RX_357(CHANNEL := CAN_CHANNEL, CAN_ID := 16#357);
(* Network 2: see the listing above *)
(* Network 3 *)
NTC_1 := RX_357.DATA[2] - 50;
NTC_2 := RX_357.DATA[3] - 50;
(* Network 4 *)
SOC_WORD := BYTE_WORD_FUNCTION(BYTE_H := RX_1E1.DATA[4], BYTE_L := RX_1E1.DATA[5]);
SOC_WORD := SOC_WORD / 10;
SOC := WORD_TO_BYTE(SOC_WORD);
(* Network 5 *)
CAPACITY_WORD := BYTE_WORD_FUNCTION(BYTE_H := RX_205.DATA[2], BYTE_L := RX_205.DATA[3]);
CAPACITY_AH := CAPACITY_WORD / 10;
CAPACITY := WORD_TO_INT(CAPACITY_AH);
TOTAL_CAPACITY_WORD := BYTE_WORD_FUNCTION(BYTE_H := RX_205.DATA[0], BYTE_L := RX_205.DATA[1]);
TOTAL_CAPACITY_AH := TOTAL_CAPACITY_WORD / 10;
TOTAL_CAPACITY := WORD_TO_INT(TOTAL_CAPACITY_AH);
(* Network 6 *)
SOH_WORD := BYTE_WORD_FUNCTION(BYTE_H := RX_205.DATA[6], BYTE_L := RX_205.DATA[7]);
SOH_WORD := SOH_WORD / 10;
SOH := WORD_TO_BYTE(SOH_WORD);
(* Network 7 *)
VOLTAGE_WORD := BYTE_WORD_FUNCTION(BYTE_H := RX_1E1.DATA[0], BYTE_L := RX_1E1.DATA[1]);
VOLTAGE_WORD := VOLTAGE_WORD / 10;
VOLTAGE := WORD_TO_INT(VOLTAGE_WORD);
(* Network 8 *)
CURRENT_WORD := BYTE_WORD_FUNCTION(BYTE_H := RX_1E1.DATA[2], BYTE_L := RX_1E1.DATA[3]);
CURRENT_WORD := CURRENT_WORD / 10;
CURRENT_WORD := CURRENT_WORD - 1000;
CURRENT := WORD_TO_INT(CURRENT_WORD);
CHARGING := CURRENT > 0;
(* Network 9 *)
POWER := VOLTAGE * CURRENT;
END_FUNCTION_BLOCK

(* POU FB_LIBRARY/RX_CAN, CFC *)
FUNCTION_BLOCK RX_CAN
(*
Created By: BHAGYESH
Date: 1-10-2023
Version: 1
Description: This function block checks the CAN data and updates the output CAN data only when it receives the new data.
*)
VAR_INPUT
	CHANNEL: BYTE;
	CAN_ID: DWORD;
END_VAR
VAR_OUTPUT
	DATA: ARRAY [0..7] OF BYTE;
	ERROR: BOOL;
END_VAR
VAR
	Rx: CAN_RX;

END_VAR
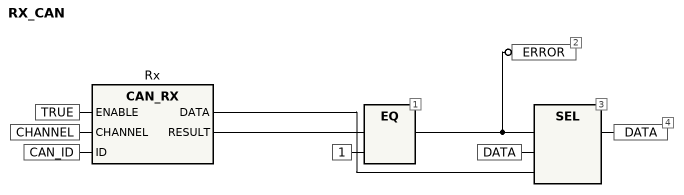
_CFC_ (* Continuous Function Chart, elements in execution order *)
#0 Rx:CAN_RX(ENABLE: TRUE, CHANNEL: CHANNEL, ID: CAN_ID)
#1 EQ(#0.RESULT, 1)
#2 ERROR <= NOT #1
#3 SEL(#1, DATA, #0.DATA)
#4 DATA <= #3
_END_CFC_
(* the same logic as Structured Text *)
Rx(ENABLE := TRUE, CHANNEL := CHANNEL, ID := CAN_ID);
ERROR := NOT (Rx.RESULT = 1);
DATA := SEL(Rx.RESULT = 1, DATA, Rx.DATA);
END_FUNCTION_BLOCK

(* POU FUNCTIONS/BYTE_WORD_FUNCTION, ST *)
FUNCTION BYTE_WORD_FUNCTION : WORD
(*
Created by: Bhagyesh Unadkat
Date: 29-03-24
Version: 1
Updated by:
Update date:
Description: This block merges Two bytes of data into WORD data.
*)
VAR_INPUT
	BYTE_H: BYTE;
	BYTE_L: BYTE;
END_VAR
VAR
	MSB: WORD;
END_VAR
MSB:= BYTE_H * 256;
BYTE_WORD_FUNCTION:= MSB + BYTE_L;
END_FUNCTION

(* POU PROGRAM_FBs/CLN_BATTERY_SELECTION, LD *)
FUNCTION_BLOCK CLN_BATTERY_SELECTION
(*
Created BY: Adiga
Date: 25-01-24
Version: 1
      
*)

VAR_INPUT
	BAT_SOC: BYTE;
	BAT_SOH: BYTE;
	BAT_POWER: INT;
	BAT_NTC1: BYTE;
	BAT_NTC2: BYTE;
	BAT_CAN_ERROR: BOOL;
	BATTERY_CAPACITY_WORD: WORD;
	BAT_CURRENT: INT;
END_VAR
VAR_OUTPUT
	LOW_SOC: BOOL;
END_VAR
VAR
	RTRIG_B1: R_TRIG;
	RTRIG_B2: R_TRIG;
	BAT_1: BOOL;
	BAT_2: BOOL;
	SOC_INT: INT;
	SOC_MAP: INT;
	SOC: BYTE;

	TON1: TON;
	TON2: TON;
END_VAR
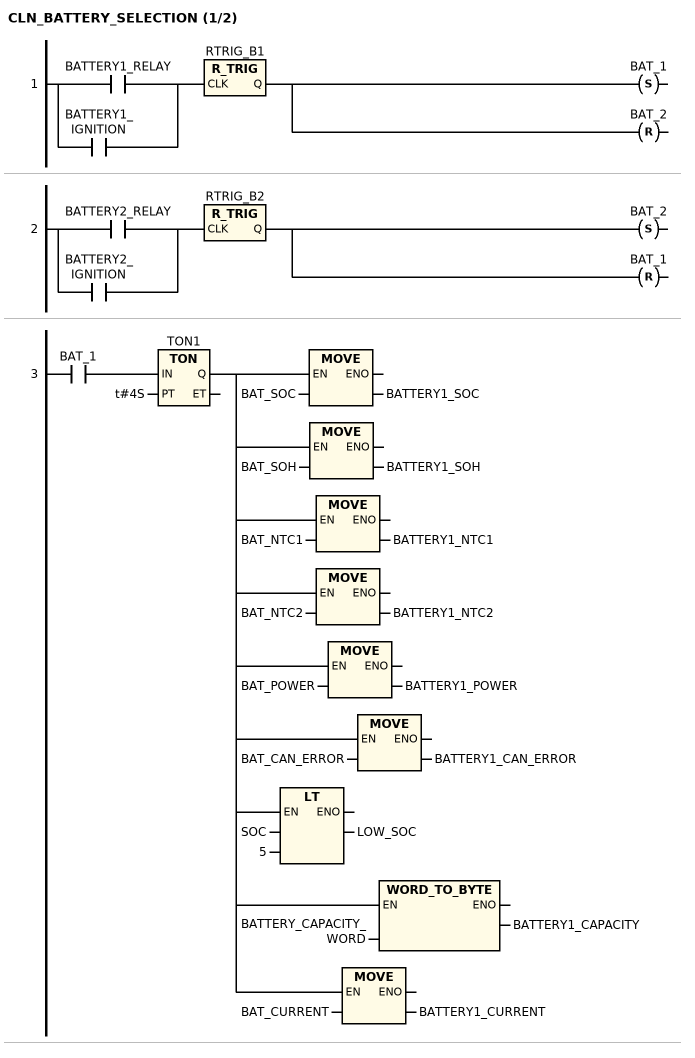
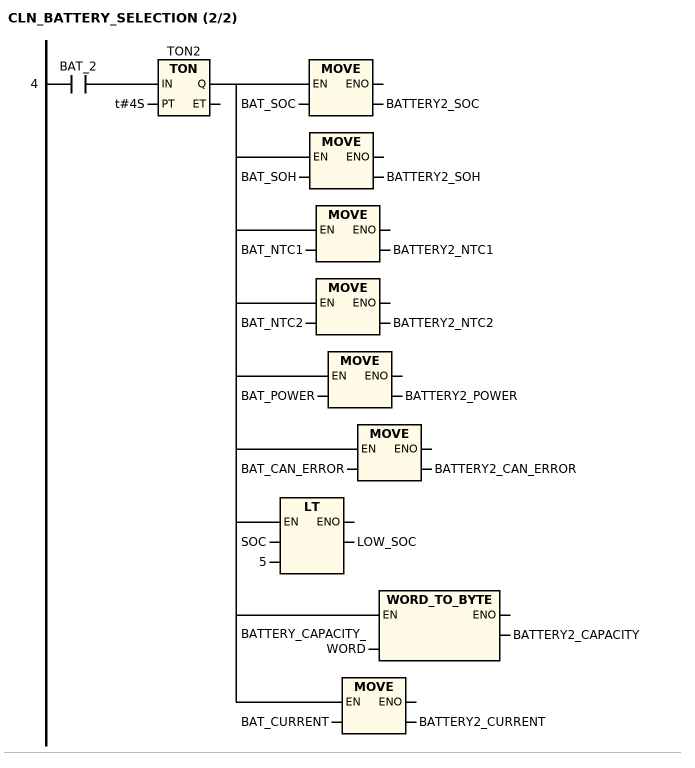
_LD_ (* Ladder Diagram *)
NETWORK 1
	{ [BATTERY1_RELAY] | [BATTERY1_IGNITION] } - RTRIG_B1:R_TRIG(CLK: *) --- (S BAT_1) (R BAT_2)
NETWORK 2
	{ [BATTERY2_RELAY] | [BATTERY2_IGNITION] } - RTRIG_B2:R_TRIG(CLK: *) --- (S BAT_2) (R BAT_1)
NETWORK 3
	[BAT_1] - TON1:TON(IN: *, PT: t#4S)
		EN --- MOVE(BAT_SOC) => BATTERY1_SOC
		EN --- MOVE(BAT_SOH) => BATTERY1_SOH
		EN --- MOVE(BAT_NTC1) => BATTERY1_NTC1
		EN --- MOVE(BAT_NTC2) => BATTERY1_NTC2
		EN --- MOVE(BAT_POWER) => BATTERY1_POWER
		EN --- MOVE(BAT_CAN_ERROR) => BATTERY1_CAN_ERROR
		EN --- LT(SOC, 5) => LOW_SOC
		EN --- WORD_TO_BYTE(BATTERY_CAPACITY_WORD) => BATTERY1_CAPACITY
		EN --- MOVE(BAT_CURRENT) => BATTERY1_CURRENT
NETWORK 4
	[BAT_2] - TON2:TON(IN: *, PT: t#4S)
		EN --- MOVE(BAT_SOC) => BATTERY2_SOC
		EN --- MOVE(BAT_SOH) => BATTERY2_SOH
		EN --- MOVE(BAT_NTC1) => BATTERY2_NTC1
		EN --- MOVE(BAT_NTC2) => BATTERY2_NTC2
		EN --- MOVE(BAT_POWER) => BATTERY2_POWER
		EN --- MOVE(BAT_CAN_ERROR) => BATTERY2_CAN_ERROR
		EN --- LT(SOC, 5) => LOW_SOC
		EN --- WORD_TO_BYTE(BATTERY_CAPACITY_WORD) => BATTERY2_CAPACITY
		EN --- MOVE(BAT_CURRENT) => BATTERY2_CURRENT
_END_LD_
(* the same logic as Structured Text *)
(* Network 1 *)
RTRIG_B1(CLK := BATTERY1_RELAY OR BATTERY1_IGNITION);
IF RTRIG_B1.Q THEN BAT_1 := TRUE; BAT_2 := FALSE; END_IF;
(* Network 2 *)
RTRIG_B2(CLK := BATTERY2_RELAY OR BATTERY2_IGNITION);
IF RTRIG_B2.Q THEN BAT_2 := TRUE; BAT_1 := FALSE; END_IF;
(* Network 3 *)
TON1(IN := BAT_1, PT := t#4S);
IF TON1.Q THEN
	BATTERY1_SOC := BAT_SOC;
	BATTERY1_SOH := BAT_SOH;
	BATTERY1_NTC1 := BAT_NTC1;
	BATTERY1_NTC2 := BAT_NTC2;
	BATTERY1_POWER := BAT_POWER;
	BATTERY1_CAN_ERROR := BAT_CAN_ERROR;
	LOW_SOC := SOC < 5;
	BATTERY1_CAPACITY := WORD_TO_BYTE(BATTERY_CAPACITY_WORD);
	BATTERY1_CURRENT := BAT_CURRENT;
END_IF;
(* Network 4 *)
TON2(IN := BAT_2, PT := t#4S);
IF TON2.Q THEN
	BATTERY2_SOC := BAT_SOC;
	BATTERY2_SOH := BAT_SOH;
	BATTERY2_NTC1 := BAT_NTC1;
	BATTERY2_NTC2 := BAT_NTC2;
	BATTERY2_POWER := BAT_POWER;
	BATTERY2_CAN_ERROR := BAT_CAN_ERROR;
	LOW_SOC := SOC < 5;
	BATTERY2_CAPACITY := WORD_TO_BYTE(BATTERY_CAPACITY_WORD);
	BATTERY2_CURRENT := BAT_CURRENT;
END_IF;
END_FUNCTION_BLOCK

(* POU PROGRAM_FBs/CLN_CHARGING, LD *)
FUNCTION_BLOCK CLN_CHARGING
(*
THIS BLOCK IS COMPATIBLE FOR 2X CLN BATTERIES0

Created BY: Adiga
Date: 25-01-24
UPDATED :14-03-25
Version: 4
1.DUAL BATTERY CAHRGING BLOCK ONLY FOR CLN
2.UPDATED THE BLOCK FOR CHARGING WITH AND WITHOUT IGN ON
3.ADDED BATTERY CAN ERROR CODITION TO CHARGE
4.ADDED TIMER BEFORE SWITCHING BATTRY BELAY.
.
*)

VAR_INPUT
	CHANNEL: BYTE;
	CHARGER_IN: BOOL;
	IGN_KEY: BOOL;
	BAT1_IGN: BOOL;
	BAT2_IGN: BOOL;
	SOC1: BYTE;
	SOC2: BYTE;
	BAT_CAN_ERROR1: BOOL;
	BAT_CAN_ERROR2: BOOL;
	BATTERY_CHARGING: BOOL;
END_VAR

VAR_OUTPUT
	RELAY_BAT1: BOOL;
	RELAY_BAT2: BOOL;
	BLUE_LED_OUT: BOOL;
	ERROR: BOOL;
	BUZZER_ON: BOOL;
	CHARGING1: BOOL;
	CHARGING2: BOOL;
END_VAR

VAR
	CHARGE_1: BOOL;
	BAT_1_FULL: BOOL;
	BAT_2_FULL: BOOL;
	T1: TON;
	T2: TON;
	T3: TON;
	IGNITION_OFF: BOOL;
	BAT_1_80: BOOL;
	BAT_2_80: BOOL;
	FTRIG1: F_TRIG;
	TIMER5: TON;
	T4: TON;
	T5: TON;
	CHARGING_2: BLINK;
	CHARGING_1: BLINK;
END_VAR
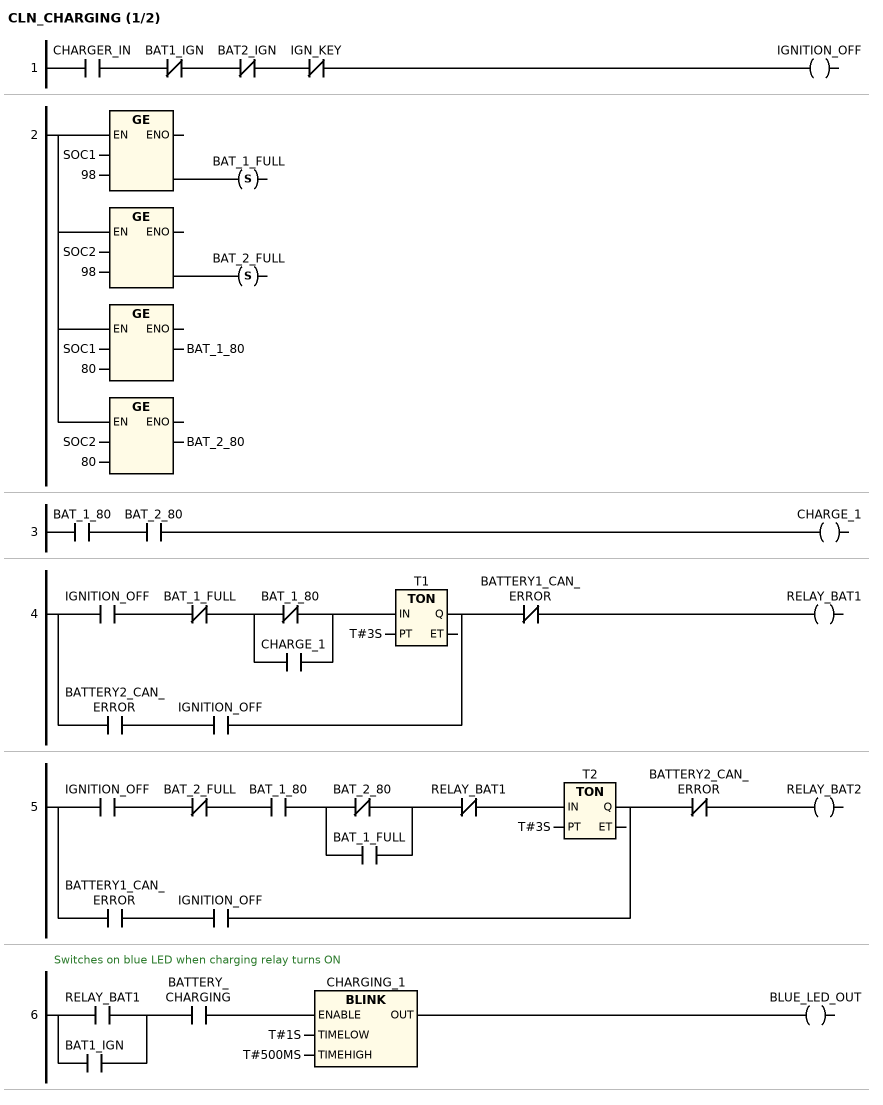
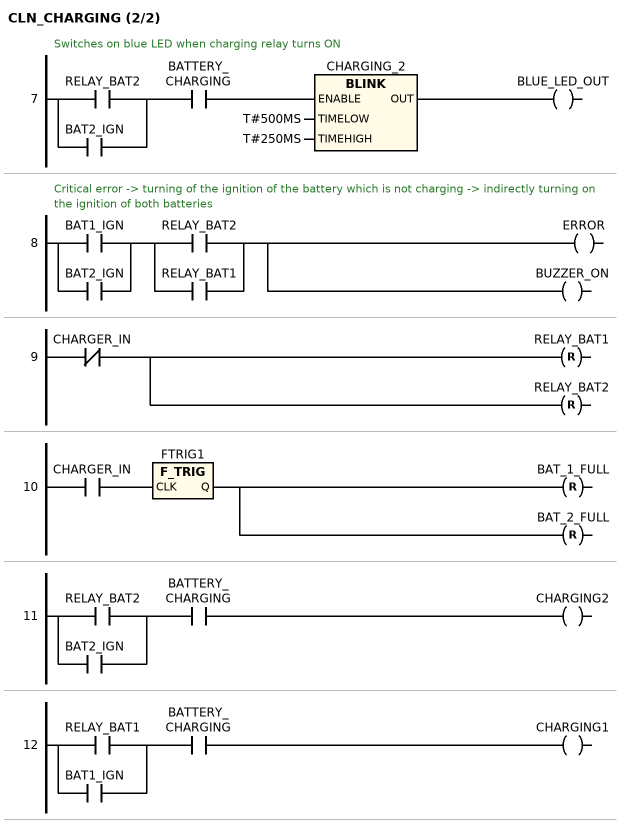
_LD_ (* Ladder Diagram *)
NETWORK 1
	[CHARGER_IN] - [/BAT1_IGN] - [/BAT2_IGN] - [/IGN_KEY] --- (IGNITION_OFF)
NETWORK 2
	*
		EN --- GE(SOC1, 98) => S BAT_1_FULL
		EN --- GE(SOC2, 98) => S BAT_2_FULL
		EN --- GE(SOC1, 80) => BAT_1_80
		EN --- GE(SOC2, 80) => BAT_2_80
NETWORK 3
	[BAT_1_80] - [BAT_2_80] --- (CHARGE_1)
NETWORK 4
	{ [IGNITION_OFF] - [/BAT_1_FULL] - { [/BAT_1_80] | [CHARGE_1] } - T1:TON(IN: *, PT: T#3S) | [BATTERY2_CAN_ERROR] - [IGNITION_OFF] } - [/BATTERY1_CAN_ERROR] --- (RELAY_BAT1)
NETWORK 5
	{ [IGNITION_OFF] - [/BAT_2_FULL] - [BAT_1_80] - { [/BAT_2_80] | [BAT_1_FULL] } - [/RELAY_BAT1] - T2:TON(IN: *, PT: T#3S) | [BATTERY1_CAN_ERROR] - [IGNITION_OFF] } - [/BATTERY2_CAN_ERROR] --- (RELAY_BAT2)
NETWORK 6 (* Switches on blue LED when charging relay turns ON *)
	{ [RELAY_BAT1] | [BAT1_IGN] } - [BATTERY_CHARGING] - CHARGING_1:BLINK(ENABLE: *, TIMELOW: T#1S, TIMEHIGH: T#500MS) --- (BLUE_LED_OUT)
NETWORK 7 (* Switches on blue LED when charging relay turns ON *)
	{ [RELAY_BAT2] | [BAT2_IGN] } - [BATTERY_CHARGING] - CHARGING_2:BLINK(ENABLE: *, TIMELOW: T#500MS, TIMEHIGH: T#250MS) --- (BLUE_LED_OUT)
NETWORK 8 (* Critical error -> turning of the ignition of the battery which is not charging -> indirectly turning on the ignition of both batteries *)
	{ [BAT1_IGN] | [BAT2_IGN] } - { [RELAY_BAT2] | [RELAY_BAT1] } --- (ERROR) (BUZZER_ON)
NETWORK 9
	[/CHARGER_IN] --- (R RELAY_BAT1) (R RELAY_BAT2)
NETWORK 10
	[CHARGER_IN] - FTRIG1:F_TRIG(CLK: *) --- (R BAT_1_FULL) (R BAT_2_FULL)
NETWORK 11
	{ [RELAY_BAT2] | [BAT2_IGN] } - [BATTERY_CHARGING] --- (CHARGING2)
NETWORK 12
	{ [RELAY_BAT1] | [BAT1_IGN] } - [BATTERY_CHARGING] --- (CHARGING1)
_END_LD_
(* the same logic as Structured Text *)
(* Network 1 *)
IGNITION_OFF := CHARGER_IN AND NOT BAT1_IGN AND NOT BAT2_IGN AND NOT IGN_KEY;
(* Network 2 *)
IF SOC1 >= 98 THEN BAT_1_FULL := TRUE; END_IF;
IF SOC2 >= 98 THEN BAT_2_FULL := TRUE; END_IF;
BAT_1_80 := SOC1 >= 80;
BAT_2_80 := SOC2 >= 80;
(* Network 3 *)
CHARGE_1 := BAT_1_80 AND BAT_2_80;
(* Network 4 *)
T1(IN := IGNITION_OFF AND NOT BAT_1_FULL AND (NOT BAT_1_80 OR CHARGE_1), PT := T#3S);
RELAY_BAT1 := (T1.Q OR BATTERY2_CAN_ERROR AND IGNITION_OFF) AND NOT BATTERY1_CAN_ERROR;
(* Network 5 *)
T2(IN := IGNITION_OFF AND NOT BAT_2_FULL AND BAT_1_80 AND (NOT BAT_2_80 OR BAT_1_FULL) AND NOT RELAY_BAT1, PT := T#3S);
RELAY_BAT2 := (T2.Q OR BATTERY1_CAN_ERROR AND IGNITION_OFF) AND NOT BATTERY2_CAN_ERROR;
(* Network 6: Switches on blue LED when charging relay turns ON *)
CHARGING_1(ENABLE := (RELAY_BAT1 OR BAT1_IGN) AND BATTERY_CHARGING, TIMELOW := T#1S, TIMEHIGH := T#500MS);
BLUE_LED_OUT := CHARGING_1.OUT;
(* Network 7: Switches on blue LED when charging relay turns ON *)
CHARGING_2(ENABLE := (RELAY_BAT2 OR BAT2_IGN) AND BATTERY_CHARGING, TIMELOW := T#500MS, TIMEHIGH := T#250MS);
BLUE_LED_OUT := CHARGING_2.OUT;
(* Network 8: Critical error -> turning of the ignition of the battery which is not charging -> indirectly turning on the ignition of both batteries *)
ERROR := (BAT1_IGN OR BAT2_IGN) AND (RELAY_BAT2 OR RELAY_BAT1);
BUZZER_ON := ERROR;
(* Network 9 *)
IF NOT CHARGER_IN THEN RELAY_BAT1 := FALSE; RELAY_BAT2 := FALSE; END_IF;
(* Network 10 *)
FTRIG1(CLK := CHARGER_IN);
IF FTRIG1.Q THEN BAT_1_FULL := FALSE; BAT_2_FULL := FALSE; END_IF;
(* Network 11 *)
CHARGING2 := (RELAY_BAT2 OR BAT2_IGN) AND BATTERY_CHARGING;
(* Network 12 *)
CHARGING1 := (RELAY_BAT1 OR BAT1_IGN) AND BATTERY_CHARGING;
END_FUNCTION_BLOCK

(* POU PROGRAM_FBs/MAKERSAN_JOYSTICK, LD *)
FUNCTION_BLOCK MAKERSAN_JOYSTICK
(*
Created by: SR Karthik Raju
Date: 23-09-24
Version: 1
Updated by:
Update date:
Description: This block reads the Makersan joystick data from the CAN.
*)
VAR_INPUT
	CAN_CHANNEL: BYTE;
END_VAR
VAR_OUTPUT
	JX: INT;
	JY: INT;
	LEFT_BUTTON: BOOL;
	RIGHT_BUTTON: BOOL;
	DEADMAN: BOOL;
	AXIS_POSITION: ARRAY [0..4] OF BOOL;
	CAN_ERROR: BOOL;
END_VAR
VAR
	RX_284: RX_CAN;
	RX_184: RX_CAN;
	TON_1: TON;
	X_WORD: WORD;
	Y_WORD: WORD;
	JX_INT: INT;
	JY_INT: INT;
	JY_ORIGIN: BOOL;
	JX_ORIGIN: BOOL;
END_VAR
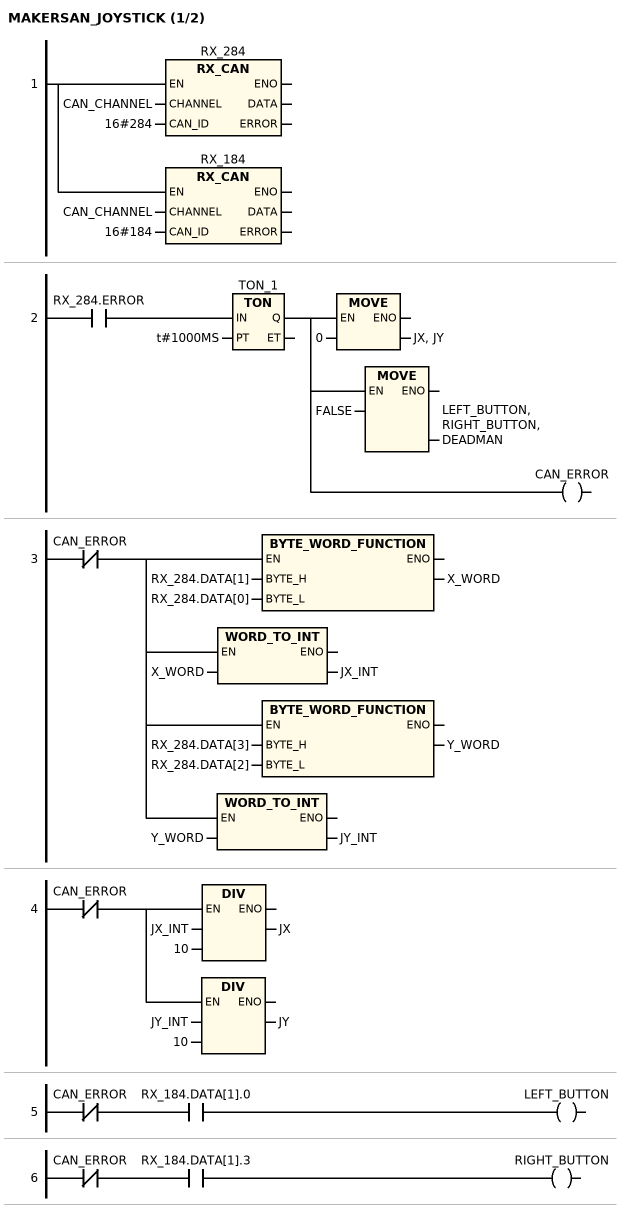
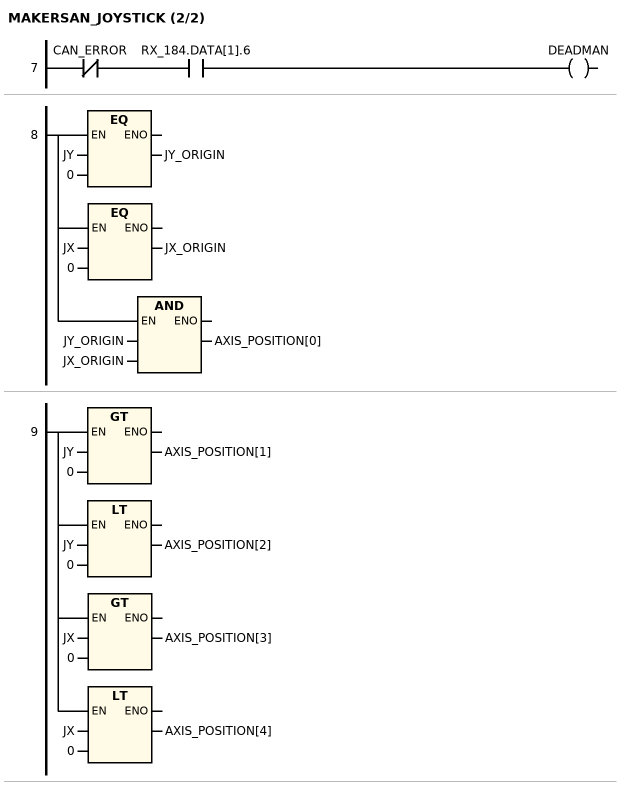
_LD_ (* Ladder Diagram *)
NETWORK 1
	*
		EN --- RX_284:RX_CAN(CHANNEL: CAN_CHANNEL, CAN_ID: 16#284)
		EN --- RX_184:RX_CAN(CHANNEL: CAN_CHANNEL, CAN_ID: 16#184)
NETWORK 2
	[RX_284.ERROR] - TON_1:TON(IN: *, PT: t#1000MS) --- (CAN_ERROR)
		EN --- MOVE(0) => JX, JY
		EN --- MOVE(FALSE) => LEFT_BUTTON, RIGHT_BUTTON, DEADMAN
NETWORK 3
	[/CAN_ERROR]
		EN --- BYTE_WORD_FUNCTION(BYTE_H: RX_284.DATA[1], BYTE_L: RX_284.DATA[0]) => X_WORD
		EN --- WORD_TO_INT(X_WORD) => JX_INT
		EN --- BYTE_WORD_FUNCTION(BYTE_H: RX_284.DATA[3], BYTE_L: RX_284.DATA[2]) => Y_WORD
		EN --- WORD_TO_INT(Y_WORD) => JY_INT
NETWORK 4
	[/CAN_ERROR]
		EN --- DIV(JX_INT, 10) => JX
		EN --- DIV(JY_INT, 10) => JY
NETWORK 5
	[/CAN_ERROR] - [RX_184.DATA[1].0] --- (LEFT_BUTTON)
NETWORK 6
	[/CAN_ERROR] - [RX_184.DATA[1].3] --- (RIGHT_BUTTON)
NETWORK 7
	[/CAN_ERROR] - [RX_184.DATA[1].6] --- (DEADMAN)
NETWORK 8
	*
		EN --- EQ(JY, 0) => JY_ORIGIN
		EN --- EQ(JX, 0) => JX_ORIGIN
		EN --- AND(JY_ORIGIN, JX_ORIGIN) => AXIS_POSITION[0]
NETWORK 9
	*
		EN --- GT(JY, 0) => AXIS_POSITION[1]
		EN --- LT(JY, 0) => AXIS_POSITION[2]
		EN --- GT(JX, 0) => AXIS_POSITION[3]
		EN --- LT(JX, 0) => AXIS_POSITION[4]
_END_LD_
(* the same logic as Structured Text *)
(* Network 1 *)
RX_284(CHANNEL := CAN_CHANNEL, CAN_ID := 16#284);
RX_184(CHANNEL := CAN_CHANNEL, CAN_ID := 16#184);
(* Network 2: see the listing above *)
(* Network 3 *)
IF NOT CAN_ERROR THEN
	X_WORD := BYTE_WORD_FUNCTION(BYTE_H := RX_284.DATA[1], BYTE_L := RX_284.DATA[0]);
	JX_INT := WORD_TO_INT(X_WORD);
	Y_WORD := BYTE_WORD_FUNCTION(BYTE_H := RX_284.DATA[3], BYTE_L := RX_284.DATA[2]);
	JY_INT := WORD_TO_INT(Y_WORD);
END_IF;
(* Network 4 *)
IF NOT CAN_ERROR THEN
	JX := JX_INT / 10;
	JY := JY_INT / 10;
END_IF;
(* Network 5 *)
LEFT_BUTTON := NOT CAN_ERROR AND RX_184.DATA[1].0;
(* Network 6 *)
RIGHT_BUTTON := NOT CAN_ERROR AND RX_184.DATA[1].3;
(* Network 7 *)
DEADMAN := NOT CAN_ERROR AND RX_184.DATA[1].6;
(* Network 8 *)
JY_ORIGIN := JY = 0;
JX_ORIGIN := JX = 0;
AXIS_POSITION[0] := JY_ORIGIN AND JX_ORIGIN;
(* Network 9 *)
AXIS_POSITION[1] := JY > 0;
AXIS_POSITION[2] := JY < 0;
AXIS_POSITION[3] := JX > 0;
AXIS_POSITION[4] := JX < 0;
END_FUNCTION_BLOCK

(* POU FB_LIBRARY/ALTERNATE, LD *)
FUNCTION_BLOCK ALTERNATE
VAR_INPUT
	IN: BOOL;
END_VAR
VAR_OUTPUT
	OUT: BOOL;
END_VAR
VAR
	S1: BOOL;
	S2: BOOL;
END_VAR
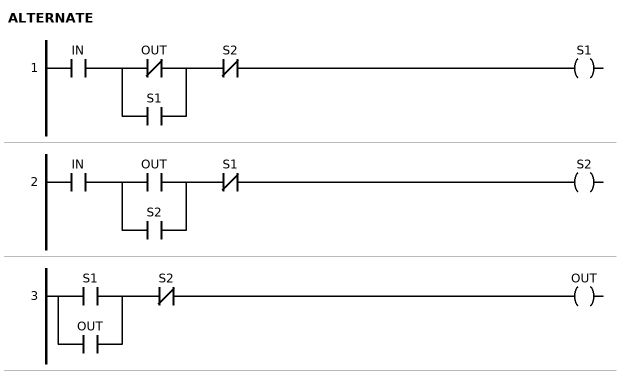
_LD_ (* Ladder Diagram *)
NETWORK 1
	[IN] - { [/OUT] | [S1] } - [/S2] --- (S1)
NETWORK 2
	[IN] - { [OUT] | [S2] } - [/S1] --- (S2)
NETWORK 3
	{ [S1] | [OUT] } - [/S2] --- (OUT)
_END_LD_
(* the same logic as Structured Text *)
(* Network 1 *)
S1 := IN AND (NOT OUT OR S1) AND NOT S2;
(* Network 2 *)
S2 := IN AND (OUT OR S2) AND NOT S1;
(* Network 3 *)
OUT := (S1 OR OUT) AND NOT S2;
END_FUNCTION_BLOCK

(* POU PROGRAM_FBs/IMU_SENSOR, LD *)
FUNCTION_BLOCK IMU_SENSOR

(*
	Created BY: Adiga
Date: 2-07-24
Version: 1
Updated BY: ADIGA
1.

*)
VAR_INPUT
END_VAR
VAR_OUTPUT
	IMY_X_OUT: BYTE;
	IMU_Y_OUT: BYTE;
	ALERT: BOOL;
END_VAR
VAR
	RX_18C: RX_CAN;
	X_ANGLE_WORD: WORD;
	X_ANGLE: INT;

	Y_ANGLE_WORD: WORD;
	Y_ANGLE: INT;

	Y_IMU: INT;
	X_IMU: INT;

	TON_IMU: TON;
	Y_ALERT: BOOL;
	PAST_TIMER: TON;
	Y_PAST: INT;
	STORE_Y_MAX: BOOL;
	X_PAST: INT;
	STORE_X_MAX: BOOL;
	STORE_Y_MIN: BOOL;
	STORE_X_MIN: BOOL;
	X_ALERT: BOOL;
	BUZZER_SOUND: BLINK;
	IMU_BUZZER: BOOL;
END_VAR
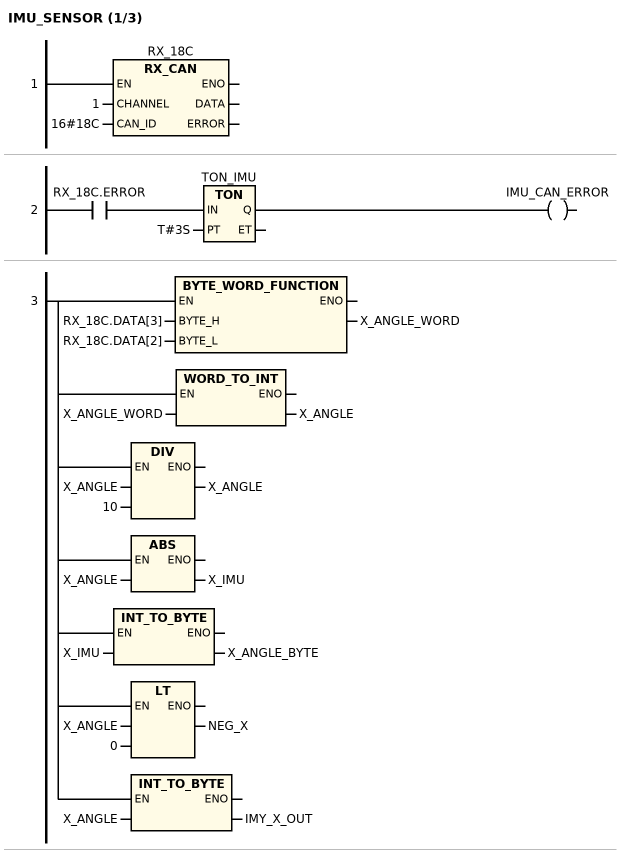
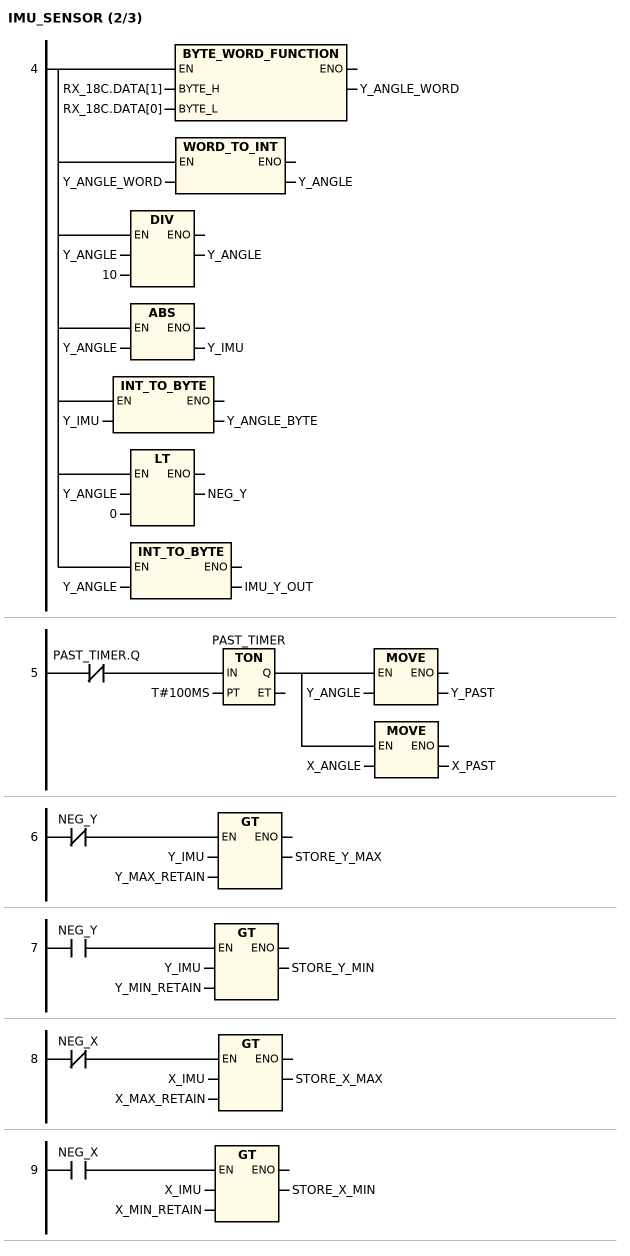
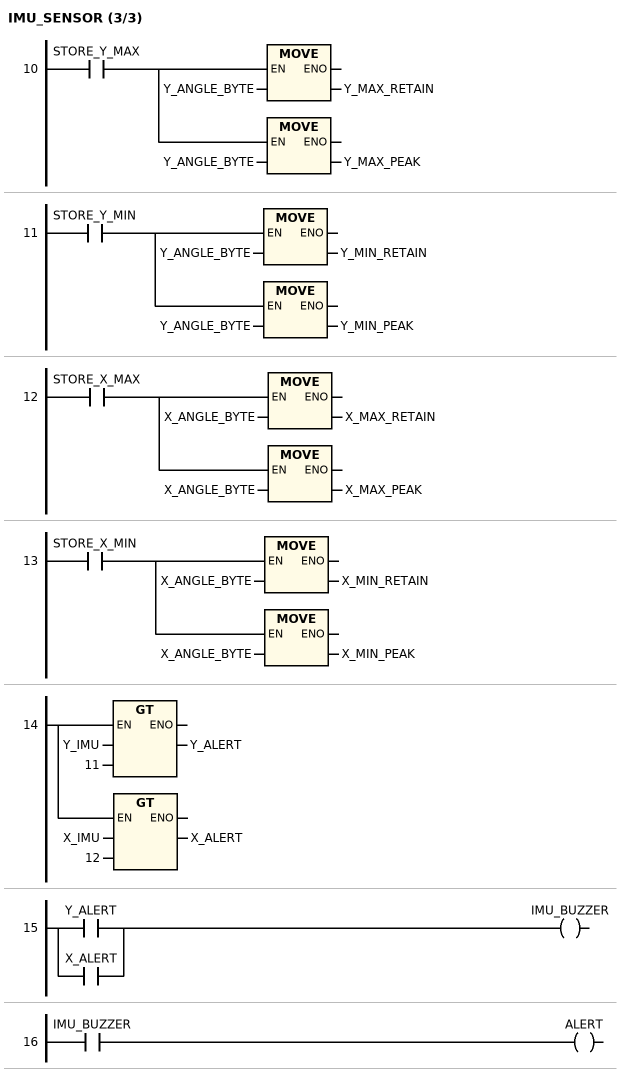
_LD_ (* Ladder Diagram *)
NETWORK 1
	*
		EN --- RX_18C:RX_CAN(CHANNEL: 1, CAN_ID: 16#18C)
NETWORK 2
	[RX_18C.ERROR] - TON_IMU:TON(IN: *, PT: T#3S) --- (IMU_CAN_ERROR)
NETWORK 3
	*
		EN --- BYTE_WORD_FUNCTION(BYTE_H: RX_18C.DATA[3], BYTE_L: RX_18C.DATA[2]) => X_ANGLE_WORD
		EN --- WORD_TO_INT(X_ANGLE_WORD) => X_ANGLE
		EN --- DIV(X_ANGLE, 10) => X_ANGLE
		EN --- ABS(X_ANGLE) => X_IMU
		EN --- INT_TO_BYTE(X_IMU) => X_ANGLE_BYTE
		EN --- LT(X_ANGLE, 0) => NEG_X
		EN --- INT_TO_BYTE(X_ANGLE) => IMY_X_OUT
NETWORK 4
	*
		EN --- BYTE_WORD_FUNCTION(BYTE_H: RX_18C.DATA[1], BYTE_L: RX_18C.DATA[0]) => Y_ANGLE_WORD
		EN --- WORD_TO_INT(Y_ANGLE_WORD) => Y_ANGLE
		EN --- DIV(Y_ANGLE, 10) => Y_ANGLE
		EN --- ABS(Y_ANGLE) => Y_IMU
		EN --- INT_TO_BYTE(Y_IMU) => Y_ANGLE_BYTE
		EN --- LT(Y_ANGLE, 0) => NEG_Y
		EN --- INT_TO_BYTE(Y_ANGLE) => IMU_Y_OUT
NETWORK 5
	[/PAST_TIMER.Q] - PAST_TIMER:TON(IN: *, PT: T#100MS)
		EN --- MOVE(Y_ANGLE) => Y_PAST
		EN --- MOVE(X_ANGLE) => X_PAST
NETWORK 6
	[/NEG_Y]
		EN --- GT(Y_IMU, Y_MAX_RETAIN) => STORE_Y_MAX
NETWORK 7
	[NEG_Y]
		EN --- GT(Y_IMU, Y_MIN_RETAIN) => STORE_Y_MIN
NETWORK 8
	[/NEG_X]
		EN --- GT(X_IMU, X_MAX_RETAIN) => STORE_X_MAX
NETWORK 9
	[NEG_X]
		EN --- GT(X_IMU, X_MIN_RETAIN) => STORE_X_MIN
NETWORK 10
	[STORE_Y_MAX]
		EN --- MOVE(Y_ANGLE_BYTE) => Y_MAX_RETAIN
		EN --- MOVE(Y_ANGLE_BYTE) => Y_MAX_PEAK
NETWORK 11
	[STORE_Y_MIN]
		EN --- MOVE(Y_ANGLE_BYTE) => Y_MIN_RETAIN
		EN --- MOVE(Y_ANGLE_BYTE) => Y_MIN_PEAK
NETWORK 12
	[STORE_X_MAX]
		EN --- MOVE(X_ANGLE_BYTE) => X_MAX_RETAIN
		EN --- MOVE(X_ANGLE_BYTE) => X_MAX_PEAK
NETWORK 13
	[STORE_X_MIN]
		EN --- MOVE(X_ANGLE_BYTE) => X_MIN_RETAIN
		EN --- MOVE(X_ANGLE_BYTE) => X_MIN_PEAK
NETWORK 14
	*
		EN --- GT(Y_IMU, 11) => Y_ALERT
		EN --- GT(X_IMU, 12) => X_ALERT
NETWORK 15
	{ [Y_ALERT] | [X_ALERT] } --- (IMU_BUZZER)
NETWORK 16
	[IMU_BUZZER] --- (ALERT)
_END_LD_
(* the same logic as Structured Text *)
(* Network 1 *)
RX_18C(CHANNEL := 1, CAN_ID := 16#18C);
(* Network 2 *)
TON_IMU(IN := RX_18C.ERROR, PT := T#3S);
IMU_CAN_ERROR := TON_IMU.Q;
(* Network 3 *)
X_ANGLE_WORD := BYTE_WORD_FUNCTION(BYTE_H := RX_18C.DATA[3], BYTE_L := RX_18C.DATA[2]);
X_ANGLE := WORD_TO_INT(X_ANGLE_WORD);
X_ANGLE := X_ANGLE / 10;
X_IMU := ABS(X_ANGLE);
X_ANGLE_BYTE := INT_TO_BYTE(X_IMU);
NEG_X := X_ANGLE < 0;
IMY_X_OUT := INT_TO_BYTE(X_ANGLE);
(* Network 4 *)
Y_ANGLE_WORD := BYTE_WORD_FUNCTION(BYTE_H := RX_18C.DATA[1], BYTE_L := RX_18C.DATA[0]);
Y_ANGLE := WORD_TO_INT(Y_ANGLE_WORD);
Y_ANGLE := Y_ANGLE / 10;
Y_IMU := ABS(Y_ANGLE);
Y_ANGLE_BYTE := INT_TO_BYTE(Y_IMU);
NEG_Y := Y_ANGLE < 0;
IMU_Y_OUT := INT_TO_BYTE(Y_ANGLE);
(* Network 5 *)
PAST_TIMER(IN := NOT PAST_TIMER.Q, PT := T#100MS);
IF PAST_TIMER.Q THEN
	Y_PAST := Y_ANGLE;
	X_PAST := X_ANGLE;
END_IF;
(* Network 6 *)
IF NOT NEG_Y THEN
	STORE_Y_MAX := Y_IMU > Y_MAX_RETAIN;
END_IF;
(* Network 7 *)
IF NEG_Y THEN
	STORE_Y_MIN := Y_IMU > Y_MIN_RETAIN;
END_IF;
(* Network 8 *)
IF NOT NEG_X THEN
	STORE_X_MAX := X_IMU > X_MAX_RETAIN;
END_IF;
(* Network 9 *)
IF NEG_X THEN
	STORE_X_MIN := X_IMU > X_MIN_RETAIN;
END_IF;
(* Network 10 *)
IF STORE_Y_MAX THEN
	Y_MAX_RETAIN := Y_ANGLE_BYTE;
	Y_MAX_PEAK := Y_ANGLE_BYTE;
END_IF;
(* Network 11 *)
IF STORE_Y_MIN THEN
	Y_MIN_RETAIN := Y_ANGLE_BYTE;
	Y_MIN_PEAK := Y_ANGLE_BYTE;
END_IF;
(* Network 12 *)
IF STORE_X_MAX THEN
	X_MAX_RETAIN := X_ANGLE_BYTE;
	X_MAX_PEAK := X_ANGLE_BYTE;
END_IF;
(* Network 13 *)
IF STORE_X_MIN THEN
	X_MIN_RETAIN := X_ANGLE_BYTE;
	X_MIN_PEAK := X_ANGLE_BYTE;
END_IF;
(* Network 14 *)
Y_ALERT := Y_IMU > 11;
X_ALERT := X_IMU > 12;
(* Network 15 *)
IMU_BUZZER := Y_ALERT OR X_ALERT;
(* Network 16 *)
ALERT := IMU_BUZZER;
END_FUNCTION_BLOCK

(* POU PROGRAM_FBs/HYDRAULIC_CONTROL, LD *)
FUNCTION_BLOCK HYDRAULIC_CONTROL
VAR_INPUT
	DEADMAN: BOOL;
END_VAR
VAR_OUTPUT
END_VAR
VAR
	HYD_SPEED: INT;
	IDLE_MODE: BOOL;
	CUTOFF: INT;
	STATISTICS: STATISTICS_INT;
	RESET_AVG: BOOL;
	T1: TON;
	TRIG_1: R_TRIG;
	T2: TON;
	RUNNING_AVG: INT:=0;
	SET_IDLE: BOOL;
	HIGH_RPM: BOOL;
	WAIT: BOOL;
	UPPER_LIMIT: INT;
	MCU_RX_6: CHARA_MCU_RX;
	MCU_TX_6: CHARA_MCU_TX;
END_VAR
VAR CONSTANT
	IDLE_SPEED: INT :=0;
	ECO_CUTOFF: INT := 70;
	POWER_CUTOFF: INT := 90;
	BUFFER: INT := 10;
	HYD_RAMP: INT:= 100;
	MCU_RAMP: BYTE := 5;
	PHASE_LIMIT: BYTE := 60;
END_VAR
